LIN {X 0,Y 251.006,Z 606.536,A -85,B 0,C 180,E1 -21636.76,E2 -21636.76} C_VEL
LIN {X 0,Y 251.097,Z 608.017,A -85,B 0,C 180,E1 -21638.716,E2 -21638.716} C_VEL
LIN {X 0,Y 252.117,Z 613.04,A -85,B 0,C 180,E1 -21642.131,E2 -21642.131} C_VEL
LIN {X 0,Y 253.267,Z 618.473,A -85,B 0,C 180,E1 -21644.407,E2 -21644.407} C_VEL
LIN {X 0,Y 253.959,Z 622.03,A -85,B 0,C 180,E1 -21645.519,E2 -21645.519} C_VEL
LIN {X 0,Y 253.455,Z 627.065,A -85,B 0,C 180,E1 -21645.978,E2 -21645.978} C_VEL
LIN {X 0,Y 248.316,Z 655.922,A -85,B 0,C 180,E1 -21647.215,E2 -21647.215} C_VEL
LIN {X 0,Y 244.438,Z 670.422,A -85,B 0,C 180,E1 -21648.052,E2 -21648.052} C_VEL
LIN {X 0,Y 239.958,Z 683.391,A -85,B 0,C 180,E1 -21649.057,E2 -21649.057} C_VEL
LIN {X 0,Y 234.475,Z 696.377,A -85,B 0,C 180,E1 -21650.438,E2 -21650.438} C_VEL
LIN {X 0,Y 229.245,Z 707.125,A -85,B 0,C 180,E1 -21651.906,E2 -21651.906} C_VEL
LIN {X 0,Y 224.326,Z 716.094,A -85,B 0,C 180,E1 -21653.47,E2 -21653.47} C_VEL
LIN {X 0,Y 218.242,Z 725.992,A -85,B 0,C 180,E1 -21655.699,E2 -21655.699} C_VEL
LIN {X 0,Y 212.71,Z 734.271,A -85,B 0,C 180,E1 -21658.087,E2 -21658.087} C_VEL
LIN {X 0,Y 207.703,Z 741.106,A -85,B 0,C 180,E1 -21660.619,E2 -21660.619} C_VEL
LIN {X 0,Y 203.369,Z 746.721,A -85,B 0,C 180,E1 -21663.305,E2 -21663.305} C_VEL
LIN {X 0,Y 199.028,Z 752.063,A -85,B 0,C 180,E1 -21666.65,E2 -21666.65} C_VEL
LIN {X 0,Y 194.978,Z 756.672,A -85,B 0,C 180,E1 -21670.798,E2 -21670.798} C_VEL
LIN {X 0,Y 193.548,Z 761.471,A -85,B 0,C 180,E1 -21673.113,E2 -21673.113} C_VEL
LIN {X 0,Y 191.946,Z 766.73,A -85,B 0,C 180,E1 -21676.232,E2 -21676.232} C_VEL
LIN {X 0,Y 190.963,Z 770.807,A -85,B 0,C 180,E1 -21679.397,E2 -21679.397} C_VEL
LIN {X 0,Y 190.551,Z 772.919,A -85,B 0,C 180,E1 -21681.516,E2 -21681.516} C_VEL
LIN {X 0,Y 190.296,Z 774.58,A -85,B 0,C 180,E1 -21683.639,E2 -21683.639} C_VEL
LIN {X 0,Y 190.173,Z 776.055,A -85,B 0,C 180,E1 -21686.202,E2 -21686.202} C_VEL
LIN {X 0,Y 190.278,Z 777.079,A -85,B 0,C 180,E1 -21690,E2 -21690} C_VEL
LIN {X 0,Y 190.186,Z 776.786,A -85,B 0,C 180,E1 -21693.856,E2 -21693.856} C_VEL
LIN {X 0,Y 190.295,Z 775.895,A -85,B 0,C 180,E1 -21696.361,E2 -21696.361} C_VEL
LIN {X 0,Y 191.029,Z 773.025,A -85,B 0,C 180,E1 -21700.6,E2 -21700.6} C_VEL
LIN {X 0,Y 192.051,Z 769.734,A -85,B 0,C 180,E1 -21703.76,E2 -21703.76} C_VEL
LIN {X 0,Y 193.68,Z 765.366,A -85,B 0,C 180,E1 -21706.875,E2 -21706.875} C_VEL
LIN {X 0,Y 195.856,Z 759.795,A -85,B 0,C 180,E1 -21709.931,E2 -21709.931} C_VEL
LIN {X 0,Y 198.526,Z 752.813,A -85,B 0,C 180,E1 -21712.917,E2 -21712.917} C_VEL
LIN {X 0,Y 201.626,Z 744.079,A -85,B 0,C 180,E1 -21715.83,E2 -21715.83} C_VEL
LIN {X 0,Y 204.75,Z 735.123,A -85,B 0,C 180,E1 -21718.161,E2 -21718.161} C_VEL
LIN {X 0,Y 207.877,Z 725.227,A -85,B 0,C 180,E1 -21720.191,E2 -21720.191} C_VEL
LIN {X 0,Y 210.84,Z 714.228,A -85,B 0,C 180,E1 -21721.948,E2 -21721.948} C_VEL
LIN {X 0,Y 213.609,Z 701.918,A -85,B 0,C 180,E1 -21723.441,E2 -21723.441} C_VEL
LIN {X 0,Y 215.784,Z 689.342,A -85,B 0,C 180,E1 -21724.534,E2 -21724.534} C_VEL
LIN {X 0,Y 217.443,Z 676.109,A -85,B 0,C 180,E1 -21725.291,E2 -21725.291} C_VEL
LIN {X 0,Y 218.773,Z 651.985,A -85,B 0,C 180,E1 -21726.098,E2 -21726.098} C_VEL
LIN {X 0,Y 220.357,Z 618.663,A -85,B 0,C 180,E1 -21727.123,E2 -21727.123} C_VEL
LIN {X 0,Y 218.124,Z 593.995,A -85,B 0,C 180,E1 -21728.604,E2 -21728.604} C_VEL
LIN {X 0,Y 217.001,Z 585.988,A -85,B 0,C 180,E1 -21729.186,E2 -21729.186} C_VEL
LIN {X 0,Y 210.259,Z 568.029,A -85,B 0,C 180,E1 -21731.555,E2 -21731.555} C_VEL
LIN {X 0,Y 203.577,Z 557.24,A -85,B 0,C 180,E1 -21733.891,E2 -21733.891} C_VEL
LIN {X 0,Y 198.403,Z 546.983,A -85,B 0,C 180,E1 -21737.699,E2 -21737.699} C_VEL
LIN {X 0,Y 194.86,Z 539.815,A -85,B 0,C 180,E1 -21740.727,E2 -21740.727} C_VEL
LIN {X 0,Y 193.325,Z 537.896,A -85,B 0,C 180,E1 -21741.83,E2 -21741.83} C_VEL
LIN {X 0,Y 192.59,Z 535.475,A -85,B 0,C 180,E1 -21742.857,E2 -21742.857} C_VEL
LIN {X 0,Y 192.605,Z 535.485,A -85,B 0,C 180,E1 -21747.059,E2 -21747.059} C_VEL
LIN {X 0,Y 192.661,Z 535.48,A -85,B 0,C 180,E1 -21751.692,E2 -21751.692} C_VEL
LIN {X 0,Y 192.681,Z 535.45,A -85,B 0,C 180,E1 -21756.346,E2 -21756.346} C_VEL
LIN {X 0,Y 192.727,Z 535.456,A -85,B 0,C 180,E1 -21761.458,E2 -21761.458} C_VEL
LIN {X 0,Y 192.847,Z 535.464,A -85,B 0,C 180,E1 -21767.37,E2 -21767.37} C_VEL
LIN {X 0,Y 193.057,Z 535.397,A -85,B 0,C 180,E1 -21771.628,E2 -21771.628} C_VEL
LIN {X 0,Y 193.26,Z 535.387,A -85,B 0,C 180,E1 -21777.916,E2 -21777.916} C_VEL
LIN {X 0,Y 193.439,Z 535.348,A -85,B 0,C 180,E1 -21780,E2 -21780} C_VEL
LIN {X 0,Y 192.973,Z 535.448,A -85,B 0,C 180,E1 -21784.178,E2 -21784.178} C_VEL
LIN {X 0,Y 193.033,Z 535.401,A -85,B 0,C 180,E1 -21788.374,E2 -21788.374} C_VEL
LIN {X 0,Y 192.797,Z 535.471,A -85,B 0,C 180,E1 -21792.634,E2 -21792.634} C_VEL
LIN {X 0,Y 192.766,Z 535.44,A -85,B 0,C 180,E1 -21796.959,E2 -21796.959} C_VEL
LIN {X 0,Y 192.638,Z 535.474,A -85,B 0,C 180,E1 -21801.398,E2 -21801.398} C_VEL
LIN {X 0,Y 192.662,Z 535.461,A -85,B 0,C 180,E1 -21804.225,E2 -21804.225} C_VEL
LIN {X 0,Y 192.648,Z 535.466,A -85,B 0,C 180,E1 -21808.893,E2 -21808.893} C_VEL
LIN {X 0,Y 192.575,Z 535.587,A -85,B 0,C 180,E1 -21813.976,E2 -21813.976} C_VEL
LIN {X 0,Y 195.327,Z 542.149,A -85,B 0,C 180,E1 -21817.711,E2 -21817.711} C_VEL
LIN {X 0,Y 198.136,Z 549.33,A -85,B 0,C 180,E1 -21821.37,E2 -21821.37} C_VEL
LIN {X 0,Y 199.487,Z 552.841,A -85,B 0,C 180,E1 -21822.961,E2 -21822.961} C_VEL
LIN {X 0,Y 206.186,Z 563.78,A -85,B 0,C 180,E1 -21825.381,E2 -21825.381} C_VEL
LIN {X 0,Y 213.008,Z 576.443,A -85,B 0,C 180,E1 -21827.668,E2 -21827.668} C_VEL
LIN {X 0,Y 218.113,Z 587.579,A -85,B 0,C 180,E1 -21829.308,E2 -21829.308} C_VEL
LIN {X 0,Y 221.247,Z 595.251,A -85,B 0,C 180,E1 -21830.294,E2 -21830.294} C_VEL
LIN {X 0,Y 221.814,Z 599.859,A -85,B 0,C 180,E1 -21830.598,E2 -21830.598} C_VEL
LIN {X 0,Y 218.375,Z 664.631,A -85,B 0,C 180,E1 -21832.595,E2 -21832.595} C_VEL
LIN {X 0,Y 216.972,Z 677.691,A -85,B 0,C 180,E1 -21833.33,E2 -21833.33} C_VEL
LIN {X 0,Y 214.979,Z 690.5,A -85,B 0,C 180,E1 -21834.43,E2 -21834.43} C_VEL
LIN {X 0,Y 212.604,Z 702.221,A -85,B 0,C 180,E1 -21835.809,E2 -21835.809} C_VEL
LIN {X 0,Y 209.799,Z 713.578,A -85,B 0,C 180,E1 -21837.591,E2 -21837.591} C_VEL
LIN {X 0,Y 206.655,Z 723.812,A -85,B 0,C 180,E1 -21839.611,E2 -21839.611} C_VEL
LIN {X 0,Y 203.821,Z 732.188,A -85,B 0,C 180,E1 -21841.699,E2 -21841.699} C_VEL
LIN {X 0,Y 200.994,Z 739.9,A -85,B 0,C 180,E1 -21844.083,E2 -21844.083} C_VEL
LIN {X 0,Y 198.07,Z 747.411,A -85,B 0,C 180,E1 -21847.027,E2 -21847.027} C_VEL
LIN {X 0,Y 195.739,Z 753.428,A -85,B 0,C 180,E1 -21850.057,E2 -21850.057} C_VEL
LIN {X 0,Y 193.716,Z 758.18,A -85,B 0,C 180,E1 -21853.128,E2 -21853.128} C_VEL
LIN {X 0,Y 192.194,Z 761.808,A -85,B 0,C 180,E1 -21856.25,E2 -21856.25} C_VEL
LIN {X 0,Y 191.192,Z 764.418,A -85,B 0,C 180,E1 -21859.409,E2 -21859.409} C_VEL
LIN {X 0,Y 190.711,Z 765.641,A -85,B 0,C 180,E1 -21861.524,E2 -21861.524} C_VEL
LIN {X 0,Y 190.381,Z 766.46,A -85,B 0,C 180,E1 -21863.642,E2 -21863.642} C_VEL
LIN {X 0,Y 190.235,Z 766.859,A -85,B 0,C 180,E1 -21865.946,E2 -21865.946} C_VEL
LIN {X 0,Y 190.278,Z 766.481,A -85,B 0,C 180,E1 -21870,E2 -21870} C_VEL
LIN {X 0,Y 190.404,Z 765.703,A -85,B 0,C 180,E1 -21872.115,E2 -21872.115} C_VEL
LIN {X 0,Y 190.718,Z 764.501,A -85,B 0,C 180,E1 -21874.226,E2 -21874.226} C_VEL
LIN {X 0,Y 191.346,Z 761.945,A -85,B 0,C 180,E1 -21877.385,E2 -21877.385} C_VEL
LIN {X 0,Y 192.355,Z 758.383,A -85,B 0,C 180,E1 -21880.526,E2 -21880.526} C_VEL
LIN {X 0,Y 193.849,Z 753.714,A -85,B 0,C 180,E1 -21883.63,E2 -21883.63} C_VEL
LIN {X 0,Y 196.246,Z 746.703,A -85,B 0,C 180,E1 -21887.184,E2 -21887.184} C_VEL
LIN {X 0,Y 198.735,Z 739.013,A -85,B 0,C 180,E1 -21890.169,E2 -21890.169} C_VEL
LIN {X 0,Y 201.736,Z 729.422,A -85,B 0,C 180,E1 -21893.074,E2 -21893.074} C_VEL
LIN {X 0,Y 204.231,Z 720.549,A -85,B 0,C 180,E1 -21895.204,E2 -21895.204} C_VEL
LIN {X 0,Y 207.06,Z 709.544,A -85,B 0,C 180,E1 -21897.271,E2 -21897.271} C_VEL
LIN {X 0,Y 209.433,Z 698.253,A -85,B 0,C 180,E1 -21898.931,E2 -21898.931} C_VEL
LIN {X 0,Y 211.508,Z 686.162,A -85,B 0,C 180,E1 -21900.266,E2 -21900.266} C_VEL
LIN {X 0,Y 213.1,Z 672.833,A -85,B 0,C 180,E1 -21901.314,E2 -21901.314} C_VEL
LIN {X 0,Y 214.137,Z 659.825,A -85,B 0,C 180,E1 -21901.951,E2 -21901.951} C_VEL
LIN {X 0,Y 217.094,Z 596.079,A -85,B 0,C 180,E1 -21903.944,E2 -21903.944} C_VEL
LIN {X 0,Y 215.869,Z 587.883,A -85,B 0,C 180,E1 -21904.501,E2 -21904.501} C_VEL
LIN {X 0,Y 210.833,Z 575.542,A -85,B 0,C 180,E1 -21906.003,E2 -21906.003} C_VEL
LIN {X 0,Y 204.574,Z 562.896,A -85,B 0,C 180,E1 -21907.9,E2 -21907.9} C_VEL
LIN {X 0,Y 198.85,Z 552.42,A -85,B 0,C 180,E1 -21909.753,E2 -21909.753} C_VEL
LIN {X 0,Y 196.161,Z 544.735,A -85,B 0,C 180,E1 -21913.074,E2 -21913.074} C_VEL
LIN {X 0,Y 195.594,Z 544.317,A -85,B 0,C 180,E1 -21913.407,E2 -21913.407} C_VEL
LIN {X 0,Y 203.792,Z 567.858,A -85,B 0,C 180,E1 -21915.364,E2 -21915.364} C_VEL
LIN {X 0,Y 200.422,Z 631.067,A -85,B 0,C 180,E1 -21918.682,E2 -21918.682} C_VEL
LIN {X 0,Y 199.667,Z 643.626,A -85,B 0,C 180,E1 -21919.7,E2 -21919.7} C_VEL
LIN {X 0,Y 198.409,Z 656.384,A -85,B 0,C 180,E1 -21921.095,E2 -21921.095} C_VEL
LIN {X 0,Y 196.986,Z 669.363,A -85,B 0,C 180,E1 -21922.982,E2 -21922.982} C_VEL
LIN {X 0,Y 195.719,Z 680.038,A -85,B 0,C 180,E1 -21924.932,E2 -21924.932} C_VEL
LIN {X 0,Y 194.244,Z 691.062,A -85,B 0,C 180,E1 -21927.438,E2 -21927.438} C_VEL
LIN {X 0,Y 192.906,Z 701.42,A -85,B 0,C 180,E1 -21930.361,E2 -21930.361} C_VEL
LIN {X 0,Y 191.938,Z 709.902,A -85,B 0,C 180,E1 -21933.349,E2 -21933.349} C_VEL
LIN {X 0,Y 191.252,Z 716.415,A -85,B 0,C 180,E1 -21936.157,E2 -21936.157} C_VEL
LIN {X 0,Y 190.736,Z 722.668,A -85,B 0,C 180,E1 -21939.509,E2 -21939.509} C_VEL
LIN {X 0,Y 190.549,Z 727.537,A -85,B 0,C 180,E1 -21942.838,E2 -21942.838} C_VEL
LIN {X 0,Y 190.823,Z 731.207,A -85,B 0,C 180,E1 -21946.149,E2 -21946.149} C_VEL
LIN {X 0,Y 191.538,Z 733.793,A -85,B 0,C 180,E1 -21949.428,E2 -21949.428} C_VEL
LIN {X 0,Y 192.288,Z 734.962,A -85,B 0,C 180,E1 -21951.593,E2 -21951.593} C_VEL
LIN {X 0,Y 193.219,Z 735.671,A -85,B 0,C 180,E1 -21953.735,E2 -21953.735} C_VEL
LIN {X 0,Y 194.384,Z 735.979,A -85,B 0,C 180,E1 -21955.853,E2 -21955.853} C_VEL
LIN {X 0,Y 196.797,Z 735.588,A -85,B 0,C 180,E1 -21959.229,E2 -21959.229} C_VEL
LIN {X 0,Y 199.268,Z 734.41,A -85,B 0,C 180,E1 -21962.021,E2 -21962.021} C_VEL
LIN {X 0,Y 201.385,Z 733.053,A -85,B 0,C 180,E1 -21964.002,E2 -21964.002} C_VEL
LIN {X 0,Y 205.459,Z 729.745,A -85,B 0,C 180,E1 -21967.27,E2 -21967.27} C_VEL
LIN {X 0,Y 210.465,Z 724.746,A -85,B 0,C 180,E1 -21970.583,E2 -21970.583} C_VEL
LIN {X 0,Y 216.064,Z 718.252,A -85,B 0,C 180,E1 -21973.64,E2 -21973.64} C_VEL
LIN {X 0,Y 221.287,Z 711.186,A -85,B 0,C 180,E1 -21976.134,E2 -21976.134} C_VEL
LIN {X 0,Y 226.988,Z 702.456,A -85,B 0,C 180,E1 -21978.503,E2 -21978.503} C_VEL
LIN {X 0,Y 232.218,Z 693.181,A -85,B 0,C 180,E1 -21980.46,E2 -21980.46} C_VEL
LIN {X 0,Y 234.395,Z 688.815,A -85,B 0,C 180,E1 -21981.23,E2 -21981.23} C_VEL
LIN {X 0,Y 236.313,Z 684.404,A -85,B 0,C 180,E1 -21982.07,E2 -21982.07} C_VEL
LIN {X 0,Y 238.302,Z 677.52,A -85,B 0,C 180,E1 -21983.734,E2 -21983.734} C_VEL
LIN {X 0,Y 240.139,Z 670.289,A -85,B 0,C 180,E1 -21985.28,E2 -21985.28} C_VEL
LIN {X 0,Y 241.666,Z 665.344,A -85,B 0,C 180,E1 -21985.936,E2 -21985.936} C_VEL
LIN {X 0,Y 245.716,Z 652.137,A -85,B 0,C 180,E1 -21987.063,E2 -21987.063} C_VEL
LIN {X 0,Y 248.489,Z 640.109,A -85,B 0,C 180,E1 -21987.813,E2 -21987.813} C_VEL
LIN {X 0,Y 252.626,Z 616.909,A -85,B 0,C 180,E1 -21988.85,E2 -21988.85} C_VEL
LIN {X 0,Y 251.193,Z 614.269,A -85,B 0,C 180,E1 -21991.022,E2 -21991.022} C_VEL
LIN {X 0,Y 250.108,Z 613.02,A -85,B 0,C 180,E1 -21993.377,E2 -21993.377} C_VEL
LIN {X 0,Y 249.533,Z 613.107,A -85,B 0,C 180,E1 -21995.798,E2 -21995.798} C_VEL
LIN {X 0,Y 249.495,Z 614.676,A -85,B 0,C 180,E1 -21998.295,E2 -21998.295} C_VEL
LIN {X 0,Y 250.173,Z 619.582,A -85,B 0,C 180,E1 -22001.613,E2 -22001.613} C_VEL
LIN {X 0,Y 251.095,Z 624.646,A -85,B 0,C 180,E1 -22003.755,E2 -22003.755} C_VEL
LIN {X 0,Y 251.331,Z 626.487,A -85,B 0,C 180,E1 -22004.326,E2 -22004.326} C_VEL
LIN {X 0,Y 250.759,Z 630.367,A -85,B 0,C 180,E1 -22004.567,E2 -22004.567} C_VEL
LIN {X 0,Y 246.269,Z 654.434,A -85,B 0,C 180,E1 -22005.588,E2 -22005.588} C_VEL
LIN {X 0,Y 242.488,Z 668.206,A -85,B 0,C 180,E1 -22006.359,E2 -22006.359} C_VEL
LIN {X 0,Y 238.113,Z 680.483,A -85,B 0,C 180,E1 -22007.247,E2 -22007.247} C_VEL
LIN {X 0,Y 232.965,Z 692.693,A -85,B 0,C 180,E1 -22008.42,E2 -22008.42} C_VEL
LIN {X 0,Y 226.813,Z 704.914,A -85,B 0,C 180,E1 -22009.989,E2 -22009.989} C_VEL
LIN {X 0,Y 221.005,Z 714.949,A -85,B 0,C 180,E1 -22011.677,E2 -22011.677} C_VEL
LIN {X 0,Y 214.571,Z 724.937,A -85,B 0,C 180,E1 -22013.875,E2 -22013.875} C_VEL
LIN {X 0,Y 208.674,Z 733.174,A -85,B 0,C 180,E1 -22016.241,E2 -22016.241} C_VEL
LIN {X 0,Y 202.458,Z 741.076,A -85,B 0,C 180,E1 -22019.202,E2 -22019.202} C_VEL
LIN {X 0,Y 197.082,Z 747.344,A -85,B 0,C 180,E1 -22022.382,E2 -22022.382} C_VEL
LIN {X 0,Y 192.036,Z 752.839,A -85,B 0,C 180,E1 -22026.262,E2 -22026.262} C_VEL
LIN {X 0,Y 188.05,Z 756.968,A -85,B 0,C 180,E1 -22030.345,E2 -22030.345} C_VEL
LIN {X 0,Y 186.738,Z 761.216,A -85,B 0,C 180,E1 -22032.478,E2 -22032.478} C_VEL
LIN {X 0,Y 185.003,Z 766.487,A -85,B 0,C 180,E1 -22035.705,E2 -22035.705} C_VEL
LIN {X 0,Y 183.945,Z 770.576,A -85,B 0,C 180,E1 -22038.987,E2 -22038.987} C_VEL
LIN {X 0,Y 183.515,Z 772.699,A -85,B 0,C 180,E1 -22041.189,E2 -22041.189} C_VEL
LIN {X 0,Y 183.224,Z 774.366,A -85,B 0,C 180,E1 -22043.392,E2 -22043.392} C_VEL
LIN {X 0,Y 183.083,Z 775.99,A -85,B 0,C 180,E1 -22046.43,E2 -22046.43} C_VEL
LIN {X 0,Y 183.184,Z 776.885,A -85,B 0,C 180,E1 -22050,E2 -22050} C_VEL
LIN {X 0,Y 183.099,Z 776.682,A -85,B 0,C 180,E1 -22053.65,E2 -22053.65} C_VEL
LIN {X 0,Y 183.224,Z 775.722,A -85,B 0,C 180,E1 -22056.608,E2 -22056.608} C_VEL
LIN {X 0,Y 184.036,Z 772.863,A -85,B 0,C 180,E1 -22061.007,E2 -22061.007} C_VEL
LIN {X 0,Y 185.124,Z 769.582,A -85,B 0,C 180,E1 -22064.286,E2 -22064.286} C_VEL
LIN {X 0,Y 186.87,Z 765.228,A -85,B 0,C 180,E1 -22067.51,E2 -22067.51} C_VEL
LIN {X 0,Y 189.164,Z 759.67,A -85,B 0,C 180,E1 -22070.668,E2 -22070.668} C_VEL
LIN {X 0,Y 191.536,Z 753.891,A -85,B 0,C 180,E1 -22073.265,E2 -22073.265} C_VEL
LIN {X 0,Y 194.65,Z 745.609,A -85,B 0,C 180,E1 -22076.25,E2 -22076.25} C_VEL
LIN {X 0,Y 197.828,Z 736.995,A -85,B 0,C 180,E1 -22078.658,E2 -22078.658} C_VEL
LIN {X 0,Y 201.385,Z 726.391,A -85,B 0,C 180,E1 -22080.98,E2 -22080.98} C_VEL
LIN {X 0,Y 204.454,Z 715.807,A -85,B 0,C 180,E1 -22082.778,E2 -22082.778} C_VEL
LIN {X 0,Y 207.325,Z 703.947,A -85,B 0,C 180,E1 -22084.301,E2 -22084.301} C_VEL
LIN {X 0,Y 209.664,Z 691.635,A -85,B 0,C 180,E1 -22085.472,E2 -22085.472} C_VEL
LIN {X 0,Y 211.484,Z 678.711,A -85,B 0,C 180,E1 -22086.294,E2 -22086.294} C_VEL
LIN {X 0,Y 212.586,Z 663.23,A -85,B 0,C 180,E1 -22086.891,E2 -22086.891} C_VEL
LIN {X 0,Y 214.742,Z 619.115,A -85,B 0,C 180,E1 -22088.283,E2 -22088.283} C_VEL
LIN {X 0,Y 212.663,Z 595.341,A -85,B 0,C 180,E1 -22089.767,E2 -22089.767} C_VEL
LIN {X 0,Y 211.799,Z 588.832,A -85,B 0,C 180,E1 -22090.254,E2 -22090.254} C_VEL
LIN {X 0,Y 205.673,Z 572.134,A -85,B 0,C 180,E1 -22092.54,E2 -22092.54} C_VEL
LIN {X 0,Y 198.272,Z 560.516,A -85,B 0,C 180,E1 -22095.189,E2 -22095.189} C_VEL
LIN {X 0,Y 196.082,Z 557.012,A -85,B 0,C 180,E1 -22096.119,E2 -22096.119} C_VEL
LIN {X 0,Y 191.992,Z 548.836,A -85,B 0,C 180,E1 -22099.478,E2 -22099.478} C_VEL
LIN {X 0,Y 190.214,Z 545.178,A -85,B 0,C 180,E1 -22101.089,E2 -22101.089} C_VEL
LIN {X 0,Y 188.506,Z 542.674,A -85,B 0,C 180,E1 -22102.455,E2 -22102.455} C_VEL
LIN {X 0,Y 187.902,Z 540.804,A -85,B 0,C 180,E1 -22103.242,E2 -22103.242} C_VEL
LIN {X 0,Y 186.047,Z 538.224,A -85,B 0,C 180,E1 -22104.825,E2 -22104.825} C_VEL
LIN {X 0,Y 185.534,Z 536.37,A -85,B 0,C 180,E1 -22105.691,E2 -22105.691} C_VEL
LIN {X 0,Y 185.579,Z 536.346,A -85,B 0,C 180,E1 -22110.576,E2 -22110.576} C_VEL
LIN {X 0,Y 185.576,Z 536.336,A -85,B 0,C 180,E1 -22115.381,E2 -22115.381} C_VEL
LIN {X 0,Y 185.67,Z 536.339,A -85,B 0,C 180,E1 -22121.134,E2 -22121.134} C_VEL
LIN {X 0,Y 185.759,Z 536.344,A -85,B 0,C 180,E1 -22126.88,E2 -22126.88} C_VEL
LIN {X 0,Y 186.004,Z 536.275,A -85,B 0,C 180,E1 -22131.308,E2 -22131.308} C_VEL
LIN {X 0,Y 186.204,Z 536.266,A -85,B 0,C 180,E1 -22137.837,E2 -22137.837} C_VEL
LIN {X 0,Y 186.403,Z 536.224,A -85,B 0,C 180,E1 -22140,E2 -22140} C_VEL
LIN {X 0,Y 185.92,Z 536.327,A -85,B 0,C 180,E1 -22144.336,E2 -22144.336} C_VEL
LIN {X 0,Y 185.979,Z 536.28,A -85,B 0,C 180,E1 -22148.695,E2 -22148.695} C_VEL
LIN {X 0,Y 185.724,Z 536.347,A -85,B 0,C 180,E1 -22153.124,E2 -22153.124} C_VEL
LIN {X 0,Y 185.713,Z 536.323,A -85,B 0,C 180,E1 -22157.623,E2 -22157.623} C_VEL
LIN {X 0,Y 185.597,Z 536.341,A -85,B 0,C 180,E1 -22162.252,E2 -22162.252} C_VEL
LIN {X 0,Y 185.561,Z 536.369,A -85,B 0,C 180,E1 -22167.033,E2 -22167.033} C_VEL
LIN {X 0,Y 185.567,Z 536.472,A -85,B 0,C 180,E1 -22171.225,E2 -22171.225} C_VEL
LIN {X 0,Y 185.855,Z 537.779,A -85,B 0,C 180,E1 -22171.966,E2 -22171.966} C_VEL
LIN {X 0,Y 188.314,Z 543.037,A -85,B 0,C 180,E1 -22175.343,E2 -22175.343} C_VEL
LIN {X 0,Y 190.843,Z 549.044,A -85,B 0,C 180,E1 -22178.76,E2 -22178.76} C_VEL
LIN {X 0,Y 192.446,Z 553.126,A -85,B 0,C 180,E1 -22180.754,E2 -22180.754} C_VEL
LIN {X 0,Y 199.267,Z 563.834,A -85,B 0,C 180,E1 -22183.453,E2 -22183.453} C_VEL
LIN {X 0,Y 205.495,Z 574.879,A -85,B 0,C 180,E1 -22185.722,E2 -22185.722} C_VEL
LIN {X 0,Y 210.934,Z 585.987,A -85,B 0,C 180,E1 -22187.597,E2 -22187.597} C_VEL
LIN {X 0,Y 215.927,Z 597.982,A -85,B 0,C 180,E1 -22189.268,E2 -22189.268} C_VEL
LIN {X 0,Y 216.242,Z 600.852,A -85,B 0,C 180,E1 -22189.459,E2 -22189.459} C_VEL
LIN {X 0,Y 212.669,Z 665.3,A -85,B 0,C 180,E1 -22191.486,E2 -22191.486} C_VEL
LIN {X 0,Y 211.198,Z 678.141,A -85,B 0,C 180,E1 -22192.231,E2 -22192.231} C_VEL
LIN {X 0,Y 209.216,Z 690.349,A -85,B 0,C 180,E1 -22193.294,E2 -22193.294} C_VEL
LIN {X 0,Y 206.733,Z 702.157,A -85,B 0,C 180,E1 -22194.696,E2 -22194.696} C_VEL
LIN {X 0,Y 203.839,Z 713.573,A -85,B 0,C 180,E1 -22196.521,E2 -22196.521} C_VEL
LIN {X 0,Y 200.562,Z 723.842,A -85,B 0,C 180,E1 -22198.585,E2 -22198.585} C_VEL
LIN {X 0,Y 197.591,Z 732.246,A -85,B 0,C 180,E1 -22200.722,E2 -22200.722} C_VEL
LIN {X 0,Y 194.626,Z 739.981,A -85,B 0,C 180,E1 -22203.169,E2 -22203.169} C_VEL
LIN {X 0,Y 191.525,Z 747.52,A -85,B 0,C 180,E1 -22206.194,E2 -22206.194} C_VEL
LIN {X 0,Y 189.024,Z 753.553,A -85,B 0,C 180,E1 -22209.316,E2 -22209.316} C_VEL
LIN {X 0,Y 186.926,Z 758.319,A -85,B 0,C 180,E1 -22212.496,E2 -22212.496} C_VEL
LIN {X 0,Y 185.277,Z 761.96,A -85,B 0,C 180,E1 -22215.726,E2 -22215.726} C_VEL
LIN {X 0,Y 184.181,Z 764.583,A -85,B 0,C 180,E1 -22219.001,E2 -22219.001} C_VEL
LIN {X 0,Y 183.673,Z 765.812,A -85,B 0,C 180,E1 -22221.196,E2 -22221.196} C_VEL
LIN {X 0,Y 183.319,Z 766.641,A -85,B 0,C 180,E1 -22223.396,E2 -22223.396} C_VEL
LIN {X 0,Y 183.138,Z 767.075,A -85,B 0,C 180,E1 -22226.18,E2 -22226.18} C_VEL
LIN {X 0,Y 183.184,Z 766.681,A -85,B 0,C 180,E1 -22230,E2 -22230} C_VEL
LIN {X 0,Y 183.318,Z 765.914,A -85,B 0,C 180,E1 -22232.197,E2 -22232.197} C_VEL
LIN {X 0,Y 183.644,Z 764.717,A -85,B 0,C 180,E1 -22234.39,E2 -22234.39} C_VEL
LIN {X 0,Y 184.22,Z 762.534,A -85,B 0,C 180,E1 -22237.29,E2 -22237.29} C_VEL
LIN {X 0,Y 185.376,Z 758.624,A -85,B 0,C 180,E1 -22240.927,E2 -22240.927} C_VEL
LIN {X 0,Y 186.97,Z 753.968,A -85,B 0,C 180,E1 -22244.142,E2 -22244.142} C_VEL
LIN {X 0,Y 189.471,Z 746.974,A -85,B 0,C 180,E1 -22247.819,E2 -22247.819} C_VEL
LIN {X 0,Y 192.102,Z 739.305,A -85,B 0,C 180,E1 -22250.897,E2 -22250.897} C_VEL
LIN {X 0,Y 195.22,Z 729.734,A -85,B 0,C 180,E1 -22253.891,E2 -22253.891} C_VEL
LIN {X 0,Y 198.199,Z 719.766,A -85,B 0,C 180,E1 -22256.31,E2 -22256.31} C_VEL
LIN {X 0,Y 201.211,Z 708.54,A -85,B 0,C 180,E1 -22258.417,E2 -22258.417} C_VEL
LIN {X 0,Y 203.523,Z 697.55,A -85,B 0,C 180,E1 -22260.042,E2 -22260.042} C_VEL
LIN {X 0,Y 205.665,Z 685.088,A -85,B 0,C 180,E1 -22261.406,E2 -22261.406} C_VEL
LIN {X 0,Y 207.242,Z 672.034,A -85,B 0,C 180,E1 -22262.426,E2 -22262.426} C_VEL
LIN {X 0,Y 208.285,Z 658.961,A -85,B 0,C 180,E1 -22263.045,E2 -22263.045} C_VEL
LIN {X 0,Y 211.335,Z 597.63,A -85,B 0,C 180,E1 -22264.983,E2 -22264.983} C_VEL
LIN {X 0,Y 210.213,Z 590.16,A -85,B 0,C 180,E1 -22265.518,E2 -22265.518} C_VEL
LIN {X 0,Y 205.221,Z 578.164,A -85,B 0,C 180,E1 -22267.083,E2 -22267.083} C_VEL
LIN {X 0,Y 198.598,Z 564.635,A -85,B 0,C 180,E1 -22269.229,E2 -22269.229} C_VEL
LIN {X 0,Y 193.412,Z 555.568,A -85,B 0,C 180,E1 -22270.989,E2 -22270.989} C_VEL
LIN {X 0,Y 191.659,Z 552.418,A -85,B 0,C 180,E1 -22271.701,E2 -22271.701} C_VEL
LIN {X 0,Y 190.947,Z 550.361,A -85,B 0,C 180,E1 -22272.597,E2 -22272.597} C_VEL
LIN {X 0,Y 190.039,Z 549.424,A -85,B 0,C 180,E1 -22273.185,E2 -22273.185} C_VEL
LIN {X 0,Y 196.819,Z 569.167,A -85,B 0,C 180,E1 -22274.937,E2 -22274.937} C_VEL
LIN {X 0,Y 193.425,Z 631.842,A -85,B 0,C 180,E1 -22278.375,E2 -22278.375} C_VEL
LIN {X 0,Y 192.447,Z 645.892,A -85,B 0,C 180,E1 -22279.578,E2 -22279.578} C_VEL
LIN {X 0,Y 191.027,Z 660.034,A -85,B 0,C 180,E1 -22281.285,E2 -22281.285} C_VEL
LIN {X 0,Y 189.53,Z 672.586,A -85,B 0,C 180,E1 -22283.277,E2 -22283.277} C_VEL
LIN {X 0,Y 188.134,Z 684.169,A -85,B 0,C 180,E1 -22285.618,E2 -22285.618} C_VEL
LIN {X 0,Y 186.725,Z 694.474,A -85,B 0,C 180,E1 -22288.201,E2 -22288.201} C_VEL
LIN {X 0,Y 185.502,Z 703.812,A -85,B 0,C 180,E1 -22291.114,E2 -22291.114} C_VEL
LIN {X 0,Y 184.528,Z 712.914,A -85,B 0,C 180,E1 -22294.629,E2 -22294.629} C_VEL
LIN {X 0,Y 183.803,Z 720.01,A -85,B 0,C 180,E1 -22298.111,E2 -22298.111} C_VEL
LIN {X 0,Y 183.454,Z 726.452,A -85,B 0,C 180,E1 -22302.153,E2 -22302.153} C_VEL
LIN {X 0,Y 183.639,Z 730.563,A -85,B 0,C 180,E1 -22305.595,E2 -22305.595} C_VEL
LIN {X 0,Y 184.302,Z 733.55,A -85,B 0,C 180,E1 -22309.008,E2 -22309.008} C_VEL
LIN {X 0,Y 185.049,Z 734.959,A -85,B 0,C 180,E1 -22311.261,E2 -22311.261} C_VEL
LIN {X 0,Y 187.119,Z 736.54,A -85,B 0,C 180,E1 -22315.691,E2 -22315.691} C_VEL
LIN {X 0,Y 189.76,Z 736.558,A -85,B 0,C 180,E1 -22319.446,E2 -22319.446} C_VEL
LIN {X 0,Y 192.062,Z 735.771,A -85,B 0,C 180,E1 -22322.097,E2 -22322.097} C_VEL
LIN {X 0,Y 194.229,Z 734.7,A -85,B 0,C 180,E1 -22324.15,E2 -22324.15} C_VEL
LIN {X 0,Y 198.53,Z 731.801,A -85,B 0,C 180,E1 -22327.616,E2 -22327.616} C_VEL
LIN {X 0,Y 203.53,Z 727.493,A -85,B 0,C 180,E1 -22330.948,E2 -22330.948} C_VEL
LIN {X 0,Y 208.428,Z 722.549,A -85,B 0,C 180,E1 -22333.652,E2 -22333.652} C_VEL
LIN {X 0,Y 213.817,Z 716.397,A -85,B 0,C 180,E1 -22336.223,E2 -22336.223} C_VEL
LIN {X 0,Y 219.506,Z 708.828,A -85,B 0,C 180,E1 -22338.673,E2 -22338.673} C_VEL
LIN {X 0,Y 225.895,Z 699.043,A -85,B 0,C 180,E1 -22341.04,E2 -22341.04} C_VEL
LIN {X 0,Y 231.457,Z 689.198,A -85,B 0,C 180,E1 -22342.88,E2 -22342.88} C_VEL
LIN {X 0,Y 236.834,Z 677.705,A -85,B 0,C 180,E1 -22344.547,E2 -22344.547} C_VEL
LIN {X 0,Y 241.666,Z 665.344,A -85,B 0,C 180,E1 -22345.936,E2 -22345.936} C_VEL
LIN {X 0,Y 243.187,Z 660.245,A -85,B 0,C 180,E1 -22346.545,E2 -22346.545} C_VEL
LIN {X 0,Y 244.76,Z 652.18,A -85,B 0,C 180,E1 -22347.85,E2 -22347.85} C_VEL
LIN {X 0,Y 246.099,Z 643.883,A -85,B 0,C 180,E1 -22349.043,E2 -22349.043} C_VEL
LIN {X 0,Y 247.077,Z 638.442,A -85,B 0,C 180,E1 -22349.491,E2 -22349.491} C_VEL
LIN {X 0,Y 250.088,Z 622.285,A -85,B 0,C 180,E1 -22350.221,E2 -22350.221} C_VEL
LIN {X 0,Y 249.289,Z 620.914,A -85,B 0,C 180,E1 -22351.623,E2 -22351.623} C_VEL
LIN {X 0,Y 248.454,Z 619.883,A -85,B 0,C 180,E1 -22353.628,E2 -22353.628} C_VEL
LIN {X 0,Y 247.912,Z 620.208,A -85,B 0,C 180,E1 -22356.171,E2 -22356.171} C_VEL
LIN {X 0,Y 247.898,Z 621.634,A -85,B 0,C 180,E1 -22358.125,E2 -22358.125} C_VEL
LIN {X 0,Y 248.339,Z 626.069,A -85,B 0,C 180,E1 -22361.076,E2 -22361.076} C_VEL
LIN {X 0,Y 248.972,Z 630.487,A -85,B 0,C 180,E1 -22362.966,E2 -22362.966} C_VEL
LIN {X 0,Y 244.341,Z 653.847,A -85,B 0,C 180,E1 -22363.978,E2 -22363.978} C_VEL
LIN {X 0,Y 240.611,Z 666.877,A -85,B 0,C 180,E1 -22364.67,E2 -22364.67} C_VEL
LIN {X 0,Y 235.889,Z 679.789,A -85,B 0,C 180,E1 -22365.561,E2 -22365.561} C_VEL
LIN {X 0,Y 230.519,Z 691.858,A -85,B 0,C 180,E1 -22366.689,E2 -22366.689} C_VEL
LIN {X 0,Y 224.087,Z 703.942,A -85,B 0,C 180,E1 -22368.207,E2 -22368.207} C_VEL
LIN {X 0,Y 217.983,Z 714.061,A -85,B 0,C 180,E1 -22369.849,E2 -22369.849} C_VEL
LIN {X 0,Y 211.162,Z 723.981,A -85,B 0,C 180,E1 -22371.996,E2 -22371.996} C_VEL
LIN {X 0,Y 203.893,Z 733.46,A -85,B 0,C 180,E1 -22374.736,E2 -22374.736} C_VEL
LIN {X 0,Y 197.327,Z 741.078,A -85,B 0,C 180,E1 -22377.708,E2 -22377.708} C_VEL
LIN {X 0,Y 190.84,Z 747.931,A -85,B 0,C 180,E1 -22381.397,E2 -22381.397} C_VEL
LIN {X 0,Y 186.747,Z 751.909,A -85,B 0,C 180,E1 -22384.356,E2 -22384.356} C_VEL
LIN {X 0,Y 181.854,Z 756.211,A -85,B 0,C 180,E1 -22389.055,E2 -22389.055} C_VEL
LIN {X 0,Y 181.348,Z 756.707,A -85,B 0,C 180,E1 -22389.587,E2 -22389.587} C_VEL
LIN {X 0,Y 179.277,Z 762.857,A -85,B 0,C 180,E1 -22392.902,E2 -22392.902} C_VEL
LIN {X 0,Y 177.655,Z 767.722,A -85,B 0,C 180,E1 -22396.27,E2 -22396.27} C_VEL
LIN {X 0,Y 176.685,Z 771.454,A -85,B 0,C 180,E1 -22399.689,E2 -22399.689} C_VEL
LIN {X 0,Y 176.148,Z 774.151,A -85,B 0,C 180,E1 -22403.126,E2 -22403.126} C_VEL
LIN {X 0,Y 175.995,Z 775.925,A -85,B 0,C 180,E1 -22406.681,E2 -22406.681} C_VEL
LIN {X 0,Y 176.091,Z 776.692,A -85,B 0,C 180,E1 -22410,E2 -22410} C_VEL
LIN {X 0,Y 175.995,Z 776.6,A -85,B 0,C 180,E1 -22413.32,E2 -22413.32} C_VEL
LIN {X 0,Y 176.149,Z 775.548,A -85,B 0,C 180,E1 -22416.874,E2 -22416.874} C_VEL
LIN {X 0,Y 177.031,Z 772.7,A -85,B 0,C 180,E1 -22421.449,E2 -22421.449} C_VEL
LIN {X 0,Y 178.199,Z 769.431,A -85,B 0,C 180,E1 -22424.853,E2 -22424.853} C_VEL
LIN {X 0,Y 180.091,Z 765.09,A -85,B 0,C 180,E1 -22428.191,E2 -22428.191} C_VEL
LIN {X 0,Y 182.521,Z 759.546,A -85,B 0,C 180,E1 -22431.456,E2 -22431.456} C_VEL
LIN {X 0,Y 185.465,Z 752.61,A -85,B 0,C 180,E1 -22434.634,E2 -22434.634} C_VEL
LIN {X 0,Y 188.908,Z 743.916,A -85,B 0,C 180,E1 -22437.712,E2 -22437.712} C_VEL
LIN {X 0,Y 192.684,Z 734.035,A -85,B 0,C 180,E1 -22440.402,E2 -22440.402} C_VEL
LIN {X 0,Y 196.098,Z 723.926,A -85,B 0,C 180,E1 -22442.519,E2 -22442.519} C_VEL
LIN {X 0,Y 199.297,Z 712.728,A -85,B 0,C 180,E1 -22444.347,E2 -22444.347} C_VEL
LIN {X 0,Y 202.169,Z 701.106,A -85,B 0,C 180,E1 -22445.763,E2 -22445.763} C_VEL
LIN {X 0,Y 204.545,Z 688.329,A -85,B 0,C 180,E1 -22446.884,E2 -22446.884} C_VEL
LIN {X 0,Y 206.284,Z 674.82,A -85,B 0,C 180,E1 -22447.67,E2 -22447.67} C_VEL
LIN {X 0,Y 209.267,Z 619.978,A -85,B 0,C 180,E1 -22449.476,E2 -22449.476} C_VEL
LIN {X 0,Y 207.307,Z 596.672,A -85,B 0,C 180,E1 -22450.989,E2 -22450.989} C_VEL
LIN {X 0,Y 206.504,Z 591.153,A -85,B 0,C 180,E1 -22451.442,E2 -22451.442} C_VEL
LIN {X 0,Y 201.211,Z 576.412,A -85,B 0,C 180,E1 -22453.545,E2 -22453.545} C_VEL
LIN {X 0,Y 194.309,Z 565.414,A -85,B 0,C 180,E1 -22456.155,E2 -22456.155} C_VEL
LIN {X 0,Y 188.646,Z 556.8,A -85,B 0,C 180,E1 -22458.603,E2 -22458.603} C_VEL
LIN {X 0,Y 185.08,Z 549.647,A -85,B 0,C 180,E1 -22461.899,E2 -22461.899} C_VEL
LIN {X 0,Y 183.803,Z 547.681,A -85,B 0,C 180,E1 -22462.998,E2 -22462.998} C_VEL
LIN {X 0,Y 183.349,Z 546.303,A -85,B 0,C 180,E1 -22463.604,E2 -22463.604} C_VEL
LIN {X 0,Y 180.076,Z 540.857,A -85,B 0,C 180,E1 -22466.881,E2 -22466.881} C_VEL
LIN {X 0,Y 178.655,Z 538.068,A -85,B 0,C 180,E1 -22468.585,E2 -22468.585} C_VEL
LIN {X 0,Y 178.491,Z 537.224,A -85,B 0,C 180,E1 -22469.048,E2 -22469.048} C_VEL
LIN {X 0,Y 178.499,Z 537.225,A -85,B 0,C 180,E1 -22474.336,E2 -22474.336} C_VEL
LIN {X 0,Y 178.52,Z 537.245,A -85,B 0,C 180,E1 -22479.249,E2 -22479.249} C_VEL
LIN {X 0,Y 178.645,Z 537.205,A -85,B 0,C 180,E1 -22481.656,E2 -22481.656} C_VEL
LIN {X 0,Y 178.676,Z 537.217,A -85,B 0,C 180,E1 -22486.35,E2 -22486.35} C_VEL
LIN {X 0,Y 178.934,Z 537.157,A -85,B 0,C 180,E1 -22490.961,E2 -22490.961} C_VEL
LIN {X 0,Y 179.15,Z 537.145,A -85,B 0,C 180,E1 -22497.752,E2 -22497.752} C_VEL
LIN {X 0,Y 179.366,Z 537.1,A -85,B 0,C 180,E1 -22500.001,E2 -22500.001} C_VEL
LIN {X 0,Y 178.867,Z 537.206,A -85,B 0,C 180,E1 -22504.508,E2 -22504.508} C_VEL
LIN {X 0,Y 178.908,Z 537.161,A -85,B 0,C 180,E1 -22509.041,E2 -22509.041} C_VEL
LIN {X 0,Y 178.654,Z 537.218,A -85,B 0,C 180,E1 -22513.653,E2 -22513.653} C_VEL
LIN {X 0,Y 178.636,Z 537.228,A -85,B 0,C 180,E1 -22519.231,E2 -22519.231} C_VEL
LIN {X 0,Y 178.533,Z 537.227,A -85,B 0,C 180,E1 -22525.125,E2 -22525.125} C_VEL
LIN {X 0,Y 178.511,Z 537.302,A -85,B 0,C 180,E1 -22527.874,E2 -22527.874} C_VEL
LIN {X 0,Y 180.399,Z 541.471,A -85,B 0,C 180,E1 -22531.012,E2 -22531.012} C_VEL
LIN {X 0,Y 183.93,Z 549.716,A -85,B 0,C 180,E1 -22536.32,E2 -22536.32} C_VEL
LIN {X 0,Y 185.435,Z 553.355,A -85,B 0,C 180,E1 -22538.275,E2 -22538.275} C_VEL
LIN {X 0,Y 192.58,Z 564.308,A -85,B 0,C 180,E1 -22541.41,E2 -22541.41} C_VEL
LIN {X 0,Y 198.217,Z 573.882,A -85,B 0,C 180,E1 -22543.654,E2 -22543.654} C_VEL
LIN {X 0,Y 204.383,Z 585.894,A -85,B 0,C 180,E1 -22545.95,E2 -22545.95} C_VEL
LIN {X 0,Y 210.165,Z 599.33,A -85,B 0,C 180,E1 -22548.008,E2 -22548.008} C_VEL
LIN {X 0,Y 210.772,Z 601.199,A -85,B 0,C 180,E1 -22548.234,E2 -22548.234} C_VEL
LIN {X 0,Y 207.148,Z 664.629,A -85,B 0,C 180,E1 -22550.26,E2 -22550.26} C_VEL
LIN {X 0,Y 205.715,Z 677.151,A -85,B 0,C 180,E1 -22550.959,E2 -22550.959} C_VEL
LIN {X 0,Y 203.608,Z 689.874,A -85,B 0,C 180,E1 -22552.061,E2 -22552.061} C_VEL
LIN {X 0,Y 200.857,Z 702.558,A -85,B 0,C 180,E1 -22553.589,E2 -22553.589} C_VEL
LIN {X 0,Y 197.954,Z 713.569,A -85,B 0,C 180,E1 -22555.387,E2 -22555.387} C_VEL
LIN {X 0,Y 194.526,Z 723.872,A -85,B 0,C 180,E1 -22557.493,E2 -22557.493} C_VEL
LIN {X 0,Y 191.419,Z 732.304,A -85,B 0,C 180,E1 -22559.68,E2 -22559.68} C_VEL
LIN {X 0,Y 188.289,Z 740.062,A -85,B 0,C 180,E1 -22562.189,E2 -22562.189} C_VEL
LIN {X 0,Y 185,Z 747.629,A -85,B 0,C 180,E1 -22565.3,E2 -22565.3} C_VEL
LIN {X 0,Y 182.349,Z 753.678,A -85,B 0,C 180,E1 -22568.523,E2 -22568.523} C_VEL
LIN {X 0,Y 180.158,Z 758.458,A -85,B 0,C 180,E1 -22571.816,E2 -22571.816} C_VEL
LIN {X 0,Y 178.355,Z 762.114,A -85,B 0,C 180,E1 -22575.16,E2 -22575.16} C_VEL
LIN {X 0,Y 177.192,Z 764.748,A -85,B 0,C 180,E1 -22578.562,E2 -22578.562} C_VEL
LIN {X 0,Y 176.636,Z 765.983,A -85,B 0,C 180,E1 -22580.843,E2 -22580.843} C_VEL
LIN {X 0,Y 176.254,Z 766.821,A -85,B 0,C 180,E1 -22583.13,E2 -22583.13} C_VEL
LIN {X 0,Y 176.047,Z 767.288,A -85,B 0,C 180,E1 -22586.415,E2 -22586.415} C_VEL
LIN {X 0,Y 176.092,Z 766.88,A -85,B 0,C 180,E1 -22590,E2 -22590} C_VEL
LIN {X 0,Y 176.234,Z 766.125,A -85,B 0,C 180,E1 -22592.285,E2 -22592.285} C_VEL
LIN {X 0,Y 176.575,Z 764.934,A -85,B 0,C 180,E1 -22594.566,E2 -22594.566} C_VEL
LIN {X 0,Y 177.113,Z 763.046,A -85,B 0,C 180,E1 -22597.236,E2 -22597.236} C_VEL
LIN {X 0,Y 178.427,Z 758.865,A -85,B 0,C 180,E1 -22601.358,E2 -22601.358} C_VEL
LIN {X 0,Y 180.116,Z 754.221,A -85,B 0,C 180,E1 -22604.692,E2 -22604.692} C_VEL
LIN {X 0,Y 182.714,Z 747.243,A -85,B 0,C 180,E1 -22608.501,E2 -22608.501} C_VEL
LIN {X 0,Y 185.503,Z 739.598,A -85,B 0,C 180,E1 -22611.677,E2 -22611.677} C_VEL
LIN {X 0,Y 188.76,Z 730.046,A -85,B 0,C 180,E1 -22614.762,E2 -22614.762} C_VEL
LIN {X 0,Y 191.892,Z 720.112,A -85,B 0,C 180,E1 -22617.245,E2 -22617.245} C_VEL
LIN {X 0,Y 195.012,Z 708.918,A -85,B 0,C 180,E1 -22619.407,E2 -22619.407} C_VEL
LIN {X 0,Y 197.349,Z 698.334,A -85,B 0,C 180,E1 -22621.022,E2 -22621.022} C_VEL
LIN {X 0,Y 199.47,Z 686.835,A -85,B 0,C 180,E1 -22622.349,E2 -22622.349} C_VEL
LIN {X 0,Y 201.216,Z 673.52,A -85,B 0,C 180,E1 -22623.448,E2 -22623.448} C_VEL
LIN {X 0,Y 202.39,Z 660.24,A -85,B 0,C 180,E1 -22624.126,E2 -22624.126} C_VEL
LIN {X 0,Y 205.549,Z 597.938,A -85,B 0,C 180,E1 -22626.154,E2 -22626.154} C_VEL
LIN {X 0,Y 204.743,Z 592.879,A -85,B 0,C 180,E1 -22626.546,E2 -22626.546} C_VEL
LIN {X 0,Y 200.051,Z 581.517,A -85,B 0,C 180,E1 -22628.105,E2 -22628.105} C_VEL
LIN {X 0,Y 193.977,Z 568.941,A -85,B 0,C 180,E1 -22630.189,E2 -22630.189} C_VEL
LIN {X 0,Y 188.533,Z 559.289,A -85,B 0,C 180,E1 -22632.151,E2 -22632.151} C_VEL
LIN {X 0,Y 187.999,Z 558.792,A -85,B 0,C 180,E1 -22632.33,E2 -22632.33} C_VEL
LIN {X 0,Y 186.466,Z 558.451,A -85,B 0,C 180,E1 -22632.796,E2 -22632.796} C_VEL
LIN {X 0,Y 185.202,Z 557.001,A -85,B 0,C 180,E1 -22633.292,E2 -22633.292} C_VEL
LIN {X 0,Y 189.89,Z 570.57,A -85,B 0,C 180,E1 -22634.498,E2 -22634.498} C_VEL
LIN {X 0,Y 186.438,Z 632.053,A -85,B 0,C 180,E1 -22638.002,E2 -22638.002} C_VEL
LIN {X 0,Y 185.519,Z 645.175,A -85,B 0,C 180,E1 -22639.149,E2 -22639.149} C_VEL
LIN {X 0,Y 184.262,Z 657.697,A -85,B 0,C 180,E1 -22640.646,E2 -22640.646} C_VEL
LIN {X 0,Y 182.709,Z 670.767,A -85,B 0,C 180,E1 -22642.711,E2 -22642.711} C_VEL
LIN {X 0,Y 181.261,Z 682.671,A -85,B 0,C 180,E1 -22645.116,E2 -22645.116} C_VEL
LIN {X 0,Y 179.632,Z 694.443,A -85,B 0,C 180,E1 -22648.117,E2 -22648.117} C_VEL
LIN {X 0,Y 178.376,Z 704.021,A -85,B 0,C 180,E1 -22651.185,E2 -22651.185} C_VEL
LIN {X 0,Y 177.418,Z 712.937,A -85,B 0,C 180,E1 -22654.721,E2 -22654.721} C_VEL
LIN {X 0,Y 176.672,Z 720.299,A -85,B 0,C 180,E1 -22658.409,E2 -22658.409} C_VEL
LIN {X 0,Y 176.385,Z 726.385,A -85,B 0,C 180,E1 -22662.341,E2 -22662.341} C_VEL
LIN {X 0,Y 176.617,Z 730.935,A -85,B 0,C 180,E1 -22666.186,E2 -22666.186} C_VEL
LIN {X 0,Y 177.08,Z 733.101,A -85,B 0,C 180,E1 -22668.554,E2 -22668.554} C_VEL
LIN {X 0,Y 177.836,Z 734.924,A -85,B 0,C 180,E1 -22671.101,E2 -22671.101} C_VEL
LIN {X 0,Y 179.823,Z 736.929,A -85,B 0,C 180,E1 -22675.516,E2 -22675.516} C_VEL
LIN {X 0,Y 182.726,Z 737.368,A -85,B 0,C 180,E1 -22679.727,E2 -22679.727} C_VEL
LIN {X 0,Y 184.83,Z 736.969,A -85,B 0,C 180,E1 -22682.179,E2 -22682.179} C_VEL
LIN {X 0,Y 187.037,Z 736.186,A -85,B 0,C 180,E1 -22684.309,E2 -22684.309} C_VEL
LIN {X 0,Y 191.622,Z 733.682,A -85,B 0,C 180,E1 -22688.012,E2 -22688.012} C_VEL
LIN {X 0,Y 196.576,Z 730.031,A -85,B 0,C 180,E1 -22691.34,E2 -22691.34} C_VEL
LIN {X 0,Y 201.626,Z 725.682,A -85,B 0,C 180,E1 -22694.122,E2 -22694.122} C_VEL
LIN {X 0,Y 207.138,Z 720.128,A -85,B 0,C 180,E1 -22696.762,E2 -22696.762} C_VEL
LIN {X 0,Y 214.065,Z 711.955,A -85,B 0,C 180,E1 -22699.665,E2 -22699.665} C_VEL
LIN {X 0,Y 219.615,Z 704.458,A -85,B 0,C 180,E1 -22701.671,E2 -22701.671} C_VEL
LIN {X 0,Y 226.155,Z 694.112,A -85,B 0,C 180,E1 -22703.827,E2 -22703.827} C_VEL
LIN {X 0,Y 232.1,Z 683.132,A -85,B 0,C 180,E1 -22705.562,E2 -22705.562} C_VEL
LIN {X 0,Y 237.131,Z 671.928,A -85,B 0,C 180,E1 -22706.949,E2 -22706.949} C_VEL
LIN {X 0,Y 241.797,Z 658.873,A -85,B 0,C 180,E1 -22708.186,E2 -22708.186} C_VEL
LIN {X 0,Y 245.482,Z 645.71,A -85,B 0,C 180,E1 -22709.124,E2 -22709.124} C_VEL
LIN {X 0,Y 247.077,Z 638.442,A -85,B 0,C 180,E1 -22709.491,E2 -22709.491} C_VEL
LIN {X 0,Y 247.538,Z 635.353,A -85,B 0,C 180,E1 -22709.795,E2 -22709.795} C_VEL
LIN {X 0,Y 247.707,Z 631.789,A -85,B 0,C 180,E1 -22710.544,E2 -22710.544} C_VEL
LIN {X 0,Y 247.507,Z 628.868,A -85,B 0,C 180,E1 -22711.675,E2 -22711.675} C_VEL
LIN {X 0,Y 247.135,Z 627.172,A -85,B 0,C 180,E1 -22712.964,E2 -22712.964} C_VEL
LIN {X 0,Y 246.911,Z 626.864,A -85,B 0,C 180,E1 -22713.635,E2 -22713.635} C_VEL
LIN {X 0,Y 246.374,Z 627.135,A -85,B 0,C 180,E1 -22716.062,E2 -22716.062} C_VEL
LIN {X 0,Y 246.303,Z 628.489,A -85,B 0,C 180,E1 -22717.846,E2 -22717.846} C_VEL
LIN {X 0,Y 246.534,Z 632.459,A -85,B 0,C 180,E1 -22720.481,E2 -22720.481} C_VEL
LIN {X 0,Y 246.692,Z 634.708,A -85,B 0,C 180,E1 -22721.519,E2 -22721.519} C_VEL
LIN {X 0,Y 242.873,Z 653.036,A -85,B 0,C 180,E1 -22722.296,E2 -22722.296} C_VEL
LIN {X 0,Y 238.987,Z 666.125,A -85,B 0,C 180,E1 -22722.975,E2 -22722.975} C_VEL
LIN {X 0,Y 233.883,Z 679.354,A -85,B 0,C 180,E1 -22723.849,E2 -22723.849} C_VEL
LIN {X 0,Y 228.339,Z 691.171,A -85,B 0,C 180,E1 -22724.936,E2 -22724.936} C_VEL
LIN {X 0,Y 221.633,Z 703.32,A -85,B 0,C 180,E1 -22726.395,E2 -22726.395} C_VEL
LIN {X 0,Y 215.267,Z 713.28,A -85,B 0,C 180,E1 -22727.99,E2 -22727.99} C_VEL
LIN {X 0,Y 208.055,Z 723.148,A -85,B 0,C 180,E1 -22730.074,E2 -22730.074} C_VEL
LIN {X 0,Y 201.408,Z 731.354,A -85,B 0,C 180,E1 -22732.364,E2 -22732.364} C_VEL
LIN {X 0,Y 194.249,Z 739.201,A -85,B 0,C 180,E1 -22735.262,E2 -22735.262} C_VEL
LIN {X 0,Y 187.889,Z 745.504,A -85,B 0,C 180,E1 -22738.422,E2 -22738.422} C_VEL
LIN {X 0,Y 181.727,Z 751.005,A -85,B 0,C 180,E1 -22742.35,E2 -22742.35} C_VEL
LIN {X 0,Y 176.797,Z 754.993,A -85,B 0,C 180,E1 -22746.577,E2 -22746.577} C_VEL
LIN {X 0,Y 174.704,Z 756.446,A -85,B 0,C 180,E1 -22748.774,E2 -22748.774} C_VEL
LIN {X 0,Y 172.488,Z 762.609,A -85,B 0,C 180,E1 -22752.207,E2 -22752.207} C_VEL
LIN {X 0,Y 170.713,Z 767.484,A -85,B 0,C 180,E1 -22755.7,E2 -22755.7} C_VEL
LIN {X 0,Y 169.676,Z 771.228,A -85,B 0,C 180,E1 -22759.258,E2 -22759.258} C_VEL
LIN {X 0,Y 169.098,Z 773.937,A -85,B 0,C 180,E1 -22762.838,E2 -22762.838} C_VEL
LIN {X 0,Y 168.898,Z 775.885,A -85,B 0,C 180,E1 -22767.029,E2 -22767.029} C_VEL
LIN {X 0,Y 169.001,Z 776.499,A -85,B 0,C 180,E1 -22770,E2 -22770} C_VEL
LIN {X 0,Y 168.91,Z 776.47,A -85,B 0,C 180,E1 -22773.043,E2 -22773.043} C_VEL
LIN {X 0,Y 169.099,Z 775.374,A -85,B 0,C 180,E1 -22777.162,E2 -22777.162} C_VEL
LIN {X 0,Y 170.054,Z 772.537,A -85,B 0,C 180,E1 -22781.925,E2 -22781.925} C_VEL
LIN {X 0,Y 171.305,Z 769.28,A -85,B 0,C 180,E1 -22785.466,E2 -22785.466} C_VEL
LIN {X 0,Y 173.344,Z 764.952,A -85,B 0,C 180,E1 -22788.926,E2 -22788.926} C_VEL
LIN {X 0,Y 175.924,Z 759.422,A -85,B 0,C 180,E1 -22792.303,E2 -22792.303} C_VEL
LIN {X 0,Y 179,Z 752.507,A -85,B 0,C 180,E1 -22795.587,E2 -22795.587} C_VEL
LIN {X 0,Y 182.632,Z 743.835,A -85,B 0,C 180,E1 -22798.751,E2 -22798.751} C_VEL
LIN {X 0,Y 186.591,Z 733.981,A -85,B 0,C 180,E1 -22801.506,E2 -22801.506} C_VEL
LIN {X 0,Y 190.142,Z 723.912,A -85,B 0,C 180,E1 -22803.67,E2 -22803.67} C_VEL
LIN {X 0,Y 193.484,Z 712.755,A -85,B 0,C 180,E1 -22805.532,E2 -22805.532} C_VEL
LIN {X 0,Y 196.459,Z 701.2,A -85,B 0,C 180,E1 -22806.972,E2 -22806.972} C_VEL
LIN {X 0,Y 198.913,Z 688.562,A -85,B 0,C 180,E1 -22808.111,E2 -22808.111} C_VEL
LIN {X 0,Y 200.722,Z 675.258,A -85,B 0,C 180,E1 -22808.906,E2 -22808.906} C_VEL
LIN {X 0,Y 202.437,Z 647.276,A -85,B 0,C 180,E1 -22809.876,E2 -22809.876} C_VEL
LIN {X 0,Y 203.838,Z 620.415,A -85,B 0,C 180,E1 -22810.764,E2 -22810.764} C_VEL
LIN {X 0,Y 202.051,Z 598.05,A -85,B 0,C 180,E1 -22812.272,E2 -22812.272} C_VEL
LIN {X 0,Y 201.425,Z 593.776,A -85,B 0,C 180,E1 -22812.644,E2 -22812.644} C_VEL
LIN {X 0,Y 196.708,Z 580.555,A -85,B 0,C 180,E1 -22814.633,E2 -22814.633} C_VEL
LIN {X 0,Y 190.377,Z 570.258,A -85,B 0,C 180,E1 -22817.172,E2 -22817.172} C_VEL
LIN {X 0,Y 184.097,Z 560.886,A -85,B 0,C 180,E1 -22819.957,E2 -22819.957} C_VEL
LIN {X 0,Y 181.317,Z 556.781,A -85,B 0,C 180,E1 -22821.376,E2 -22821.376} C_VEL
LIN {X 0,Y 178.831,Z 551.95,A -85,B 0,C 180,E1 -22823.879,E2 -22823.879} C_VEL
LIN {X 0,Y 175.303,Z 545.627,A -85,B 0,C 180,E1 -22827.726,E2 -22827.726} C_VEL
LIN {X 0,Y 173.527,Z 542.237,A -85,B 0,C 180,E1 -22830.025,E2 -22830.025} C_VEL
LIN {X 0,Y 171.954,Z 539.999,A -85,B 0,C 180,E1 -22831.965,E2 -22831.965} C_VEL
LIN {X 0,Y 171.411,Z 538.124,A -85,B 0,C 180,E1 -22833.192,E2 -22833.192} C_VEL
LIN {X 0,Y 171.449,Z 538.111,A -85,B 0,C 180,E1 -22838.351,E2 -22838.351} C_VEL
LIN {X 0,Y 171.574,Z 538.096,A -85,B 0,C 180,E1 -22840.872,E2 -22840.872} C_VEL
LIN {X 0,Y 171.588,Z 538.088,A -85,B 0,C 180,E1 -22845.774,E2 -22845.774} C_VEL
LIN {X 0,Y 171.869,Z 538.038,A -85,B 0,C 180,E1 -22850.587,E2 -22850.587} C_VEL
LIN {X 0,Y 171.82,Z 538.08,A -85,B 0,C 180,E1 -22855.308,E2 -22855.308} C_VEL
LIN {X 0,Y 172.329,Z 537.976,A -85,B 0,C 180,E1 -22860.001,E2 -22860.001} C_VEL
LIN {X 0,Y 171.815,Z 538.082,A -85,B 0,C 180,E1 -22864.693,E2 -22864.693} C_VEL
LIN {X 0,Y 171.845,Z 538.042,A -85,B 0,C 180,E1 -22869.416,E2 -22869.416} C_VEL
LIN {X 0,Y 171.573,Z 538.09,A -85,B 0,C 180,E1 -22874.228,E2 -22874.228} C_VEL
LIN {X 0,Y 171.555,Z 538.114,A -85,B 0,C 180,E1 -22879.575,E2 -22879.575} C_VEL
LIN {X 0,Y 171.455,Z 538.104,A -85,B 0,C 180,E1 -22883.878,E2 -22883.878} C_VEL
LIN {X 0,Y 172.702,Z 541.319,A -85,B 0,C 180,E1 -22886.593,E2 -22886.593} C_VEL
LIN {X 0,Y 173.52,Z 542.539,A -85,B 0,C 180,E1 -22887.761,E2 -22887.761} C_VEL
LIN {X 0,Y 176.359,Z 548.953,A -85,B 0,C 180,E1 -22892.549,E2 -22892.549} C_VEL
LIN {X 0,Y 178.294,Z 553.436,A -85,B 0,C 180,E1 -22895.378,E2 -22895.378} C_VEL
LIN {X 0,Y 182.975,Z 560.346,A -85,B 0,C 180,E1 -22897.755,E2 -22897.755} C_VEL
LIN {X 0,Y 188.475,Z 568.757,A -85,B 0,C 180,E1 -22900.276,E2 -22900.276} C_VEL
LIN {X 0,Y 194.643,Z 579.518,A -85,B 0,C 180,E1 -22902.872,E2 -22902.872} C_VEL
LIN {X 0,Y 200.24,Z 590.843,A -85,B 0,C 180,E1 -22905.073,E2 -22905.073} C_VEL
LIN {X 0,Y 205.339,Z 603.036,A -85,B 0,C 180,E1 -22906.996,E2 -22906.996} C_VEL
LIN {X 0,Y 201.624,Z 665.301,A -85,B 0,C 180,E1 -22909.025,E2 -22909.025} C_VEL
LIN {X 0,Y 200.024,Z 678.327,A -85,B 0,C 180,E1 -22909.789,E2 -22909.789} C_VEL
LIN {X 0,Y 197.835,Z 690.807,A -85,B 0,C 180,E1 -22910.91,E2 -22910.91} C_VEL
LIN {X 0,Y 194.974,Z 703.299,A -85,B 0,C 180,E1 -22912.469,E2 -22912.469} C_VEL
LIN {X 0,Y 191.73,Z 714.823,A -85,B 0,C 180,E1 -22914.416,E2 -22914.416} C_VEL
LIN {X 0,Y 188.197,Z 724.948,A -85,B 0,C 180,E1 -22916.577,E2 -22916.577} C_VEL
LIN {X 0,Y 184.597,Z 734.05,A -85,B 0,C 180,E1 -22919.072,E2 -22919.072} C_VEL
LIN {X 0,Y 180.774,Z 742.849,A -85,B 0,C 180,E1 -22922.192,E2 -22922.192} C_VEL
LIN {X 0,Y 177.884,Z 749.166,A -85,B 0,C 180,E1 -22925.057,E2 -22925.057} C_VEL
LIN {X 0,Y 174.935,Z 755.557,A -85,B 0,C 180,E1 -22928.804,E2 -22928.804} C_VEL
LIN {X 0,Y 172.668,Z 759.958,A -85,B 0,C 180,E1 -22932.226,E2 -22932.226} C_VEL
LIN {X 0,Y 171.011,Z 763.275,A -85,B 0,C 180,E1 -22935.725,E2 -22935.725} C_VEL
LIN {X 0,Y 170.224,Z 764.913,A -85,B 0,C 180,E1 -22938.087,E2 -22938.087} C_VEL
LIN {X 0,Y 169.214,Z 767.001,A -85,B 0,C 180,E1 -22942.843,E2 -22942.843} C_VEL
LIN {X 0,Y 168.932,Z 767.488,A -85,B 0,C 180,E1 -22946.835,E2 -22946.835} C_VEL
LIN {X 0,Y 169.002,Z 767.079,A -85,B 0,C 180,E1 -22950,E2 -22950} C_VEL
LIN {X 0,Y 169.152,Z 766.334,A -85,B 0,C 180,E1 -22952.381,E2 -22952.381} C_VEL
LIN {X 0,Y 169.51,Z 765.151,A -85,B 0,C 180,E1 -22954.756,E2 -22954.756} C_VEL
LIN {X 0,Y 169.987,Z 763.572,A -85,B 0,C 180,E1 -22957.125,E2 -22957.125} C_VEL
LIN {X 0,Y 171.008,Z 760.392,A -85,B 0,C 180,E1 -22960.657,E2 -22960.657} C_VEL
LIN {X 0,Y 172.605,Z 756.147,A -85,B 0,C 180,E1 -22964.14,E2 -22964.14} C_VEL
LIN {X 0,Y 174.744,Z 750.719,A -85,B 0,C 180,E1 -22967.556,E2 -22967.556} C_VEL
LIN {X 0,Y 177.412,Z 743.924,A -85,B 0,C 180,E1 -22970.886,E2 -22970.886} C_VEL
LIN {X 0,Y 180.594,Z 735.384,A -85,B 0,C 180,E1 -22974.117,E2 -22974.117} C_VEL
LIN {X 0,Y 183.565,Z 726.641,A -85,B 0,C 180,E1 -22976.734,E2 -22976.734} C_VEL
LIN {X 0,Y 186.636,Z 717.042,A -85,B 0,C 180,E1 -22979,E2 -22979} C_VEL
LIN {X 0,Y 189.588,Z 706.439,A -85,B 0,C 180,E1 -22980.953,E2 -22980.953} C_VEL
LIN {X 0,Y 191.944,Z 695.948,A -85,B 0,C 180,E1 -22982.474,E2 -22982.474} C_VEL
LIN {X 0,Y 194.075,Z 683.656,A -85,B 0,C 180,E1 -22983.832,E2 -22983.832} C_VEL
LIN {X 0,Y 195.678,Z 671.581,A -85,B 0,C 180,E1 -22984.761,E2 -22984.761} C_VEL
LIN {X 0,Y 196.805,Z 657.573,A -85,B 0,C 180,E1 -22985.411,E2 -22985.411} C_VEL
LIN {X 0,Y 199.935,Z 599.611,A -85,B 0,C 180,E1 -22987.313,E2 -22987.313} C_VEL
LIN {X 0,Y 199.262,Z 595.28,A -85,B 0,C 180,E1 -22987.663,E2 -22987.663} C_VEL
LIN {X 0,Y 193.996,Z 582.709,A -85,B 0,C 180,E1 -22989.522,E2 -22989.522} C_VEL
LIN {X 0,Y 187.644,Z 569.8,A -85,B 0,C 180,E1 -22991.866,E2 -22991.866} C_VEL
LIN {X 0,Y 187.316,Z 569.253,A -85,B 0,C 180,E1 -22991.987,E2 -22991.987} C_VEL
LIN {X 0,Y 186.202,Z 569.508,A -85,B 0,C 180,E1 -22992.295,E2 -22992.295} C_VEL
LIN {X 0,Y 185.286,Z 570.227,A -85,B 0,C 180,E1 -22992.526,E2 -22992.526} C_VEL
LIN {X 0,Y 182.752,Z 569.868,A -85,B 0,C 180,E1 -22993.307,E2 -22993.307} C_VEL
LIN {X 0,Y 181.791,Z 568.504,A -85,B 0,C 180,E1 -22993.679,E2 -22993.679} C_VEL
LIN {X 0,Y 182.95,Z 571.921,A -85,B 0,C 180,E1 -22994.028,E2 -22994.028} C_VEL
LIN {X 0,Y 179.422,Z 632.669,A -85,B 0,C 180,E1 -22997.681,E2 -22997.681} C_VEL
LIN {X 0,Y 178.429,Z 645.972,A -85,B 0,C 180,E1 -22998.906,E2 -22998.906} C_VEL
LIN {X 0,Y 177.064,Z 659.164,A -85,B 0,C 180,E1 -23000.574,E2 -23000.574} C_VEL
LIN {X 0,Y 175.494,Z 672.061,A -85,B 0,C 180,E1 -23002.719,E2 -23002.719} C_VEL
LIN {X 0,Y 174.014,Z 683.78,A -85,B 0,C 180,E1 -23005.217,E2 -23005.217} C_VEL
LIN {X 0,Y 172.516,Z 694.372,A -85,B 0,C 180,E1 -23008.021,E2 -23008.021} C_VEL
LIN {X 0,Y 171.264,Z 703.991,A -85,B 0,C 180,E1 -23011.172,E2 -23011.172} C_VEL
LIN {X 0,Y 170.397,Z 712.074,A -85,B 0,C 180,E1 -23014.455,E2 -23014.455} C_VEL
LIN {X 0,Y 169.621,Z 719.354,A -85,B 0,C 180,E1 -23018.105,E2 -23018.105} C_VEL
LIN {X 0,Y 169.322,Z 725.274,A -85,B 0,C 180,E1 -23021.803,E2 -23021.803} C_VEL
LIN {X 0,Y 169.445,Z 730.024,A -85,B 0,C 180,E1 -23025.589,E2 -23025.589} C_VEL
LIN {X 0,Y 169.871,Z 732.466,A -85,B 0,C 180,E1 -23028.061,E2 -23028.061} C_VEL
LIN {X 0,Y 170.708,Z 734.901,A -85,B 0,C 180,E1 -23031.134,E2 -23031.134} C_VEL
LIN {X 0,Y 172.52,Z 737.108,A -85,B 0,C 180,E1 -23035.326,E2 -23035.326} C_VEL
LIN {X 0,Y 175.656,Z 738.098,A -85,B 0,C 180,E1 -23039.999,E2 -23039.999} C_VEL
LIN {X 0,Y 177.597,Z 738.01,A -85,B 0,C 180,E1 -23042.267,E2 -23042.267} C_VEL
LIN {X 0,Y 179.835,Z 737.484,A -85,B 0,C 180,E1 -23044.482,E2 -23044.482} C_VEL
LIN {X 0,Y 184.755,Z 735.375,A -85,B 0,C 180,E1 -23048.504,E2 -23048.504} C_VEL
LIN {X 0,Y 189.635,Z 732.427,A -85,B 0,C 180,E1 -23051.761,E2 -23051.761} C_VEL
LIN {X 0,Y 194.793,Z 728.586,A -85,B 0,C 180,E1 -23054.628,E2 -23054.628} C_VEL
LIN {X 0,Y 200.457,Z 723.622,A -85,B 0,C 180,E1 -23057.338,E2 -23057.338} C_VEL
LIN {X 0,Y 206.557,Z 717.46,A -85,B 0,C 180,E1 -23059.892,E2 -23059.892} C_VEL
LIN {X 0,Y 213.048,Z 709.799,A -85,B 0,C 180,E1 -23062.266,E2 -23062.266} C_VEL
LIN {X 0,Y 220.089,Z 700.233,A -85,B 0,C 180,E1 -23064.527,E2 -23064.527} C_VEL
LIN {X 0,Y 226.302,Z 690.255,A -85,B 0,C 180,E1 -23066.316,E2 -23066.316} C_VEL
LIN {X 0,Y 232.302,Z 678.755,A -85,B 0,C 180,E1 -23067.923,E2 -23067.923} C_VEL
LIN {X 0,Y 236.916,Z 668.246,A -85,B 0,C 180,E1 -23069.062,E2 -23069.062} C_VEL
LIN {X 0,Y 241.489,Z 655.04,A -85,B 0,C 180,E1 -23070.172,E2 -23070.172} C_VEL
LIN {X 0,Y 244.837,Z 642.262,A -85,B 0,C 180,E1 -23070.954,E2 -23070.954} C_VEL
LIN {X 0,Y 247.735,Z 627.856,A -85,B 0,C 180,E1 -23071.616,E2 -23071.616} C_VEL
LIN {X 0,Y 246.911,Z 626.864,A -85,B 0,C 180,E1 -23073.635,E2 -23073.635} C_VEL
LIN {X 0,Y 246.54,Z 627.442,A -85,B 0,C 180,E1 -23074.527,E2 -23074.527} C_VEL
LIN {X 0,Y 245.868,Z 629.72,A -85,B 0,C 180,E1 -23075.629,E2 -23075.629} C_VEL
LIN {X 0,Y 244.797,Z 634.938,A -85,B 0,C 180,E1 -23077.498,E2 -23077.498} C_VEL
LIN {X 0,Y 244.659,Z 636.088,A -85,B 0,C 180,E1 -23078.081,E2 -23078.081} C_VEL
LIN {X 0,Y 244.762,Z 639.042,A -85,B 0,C 180,E1 -23079.975,E2 -23079.975} C_VEL
LIN {X 0,Y 244.57,Z 640.225,A -85,B 0,C 180,E1 -23080.104,E2 -23080.104} C_VEL
LIN {X 0,Y 241.064,Z 654.869,A -85,B 0,C 180,E1 -23080.713,E2 -23080.713} C_VEL
LIN {X 0,Y 236.587,Z 668.414,A -85,B 0,C 180,E1 -23081.424,E2 -23081.424} C_VEL
LIN {X 0,Y 231.092,Z 681.472,A -85,B 0,C 180,E1 -23082.306,E2 -23082.306} C_VEL
LIN {X 0,Y 225.413,Z 692.735,A -85,B 0,C 180,E1 -23083.35,E2 -23083.35} C_VEL
LIN {X 0,Y 218.749,Z 703.921,A -85,B 0,C 180,E1 -23084.699,E2 -23084.699} C_VEL
LIN {X 0,Y 210.187,Z 716.186,A -85,B 0,C 180,E1 -23086.73,E2 -23086.73} C_VEL
LIN {X 0,Y 202.79,Z 725.401,A -85,B 0,C 180,E1 -23088.818,E2 -23088.818} C_VEL
LIN {X 0,Y 193.747,Z 735.299,A -85,B 0,C 180,E1 -23091.928,E2 -23091.928} C_VEL
LIN {X 0,Y 187.536,Z 741.297,A -85,B 0,C 180,E1 -23094.489,E2 -23094.489} C_VEL
LIN {X 0,Y 180.204,Z 747.622,A -85,B 0,C 180,E1 -23098.231,E2 -23098.231} C_VEL
LIN {X 0,Y 175.468,Z 751.32,A -85,B 0,C 180,E1 -23101.274,E2 -23101.274} C_VEL
LIN {X 0,Y 170.283,Z 754.885,A -85,B 0,C 180,E1 -23105.625,E2 -23105.625} C_VEL
LIN {X 0,Y 168.113,Z 756.187,A -85,B 0,C 180,E1 -23107.899,E2 -23107.899} C_VEL
LIN {X 0,Y 165.702,Z 762.36,A -85,B 0,C 180,E1 -23111.452,E2 -23111.452} C_VEL
LIN {X 0,Y 163.794,Z 767.247,A -85,B 0,C 180,E1 -23115.082,E2 -23115.082} C_VEL
LIN {X 0,Y 162.691,Z 771.003,A -85,B 0,C 180,E1 -23118.791,E2 -23118.791} C_VEL
LIN {X 0,Y 162.022,Z 773.722,A -85,B 0,C 180,E1 -23122.523,E2 -23122.523} C_VEL
LIN {X 0,Y 161.832,Z 775.789,A -85,B 0,C 180,E1 -23127.231,E2 -23127.231} C_VEL
LIN {X 0,Y 161.913,Z 776.305,A -85,B 0,C 180,E1 -23130,E2 -23130} C_VEL
LIN {X 0,Y 161.828,Z 776.312,A -85,B 0,C 180,E1 -23132.741,E2 -23132.741} C_VEL
LIN {X 0,Y 162.026,Z 775.199,A -85,B 0,C 180,E1 -23137.477,E2 -23137.477} C_VEL
LIN {X 0,Y 163.097,Z 772.375,A -85,B 0,C 180,E1 -23142.442,E2 -23142.442} C_VEL
LIN {X 0,Y 164.443,Z 769.129,A -85,B 0,C 180,E1 -23146.128,E2 -23146.128} C_VEL
LIN {X 0,Y 166.631,Z 764.814,A -85,B 0,C 180,E1 -23149.719,E2 -23149.719} C_VEL
LIN {X 0,Y 169.372,Z 759.299,A -85,B 0,C 180,E1 -23153.215,E2 -23153.215} C_VEL
LIN {X 0,Y 172.585,Z 752.403,A -85,B 0,C 180,E1 -23156.611,E2 -23156.611} C_VEL
LIN {X 0,Y 176.432,Z 743.754,A -85,B 0,C 180,E1 -23159.862,E2 -23159.862} C_VEL
LIN {X 0,Y 180.168,Z 734.89,A -85,B 0,C 180,E1 -23162.435,E2 -23162.435} C_VEL
LIN {X 0,Y 183.861,Z 725.142,A -85,B 0,C 180,E1 -23164.651,E2 -23164.651} C_VEL
LIN {X 0,Y 187.333,Z 714.337,A -85,B 0,C 180,E1 -23166.552,E2 -23166.552} C_VEL
LIN {X 0,Y 190.597,Z 702.259,A -85,B 0,C 180,E1 -23168.142,E2 -23168.142} C_VEL
LIN {X 0,Y 193.256,Z 689.531,A -85,B 0,C 180,E1 -23169.355,E2 -23169.355} C_VEL
LIN {X 0,Y 195.142,Z 676.777,A -85,B 0,C 180,E1 -23170.156,E2 -23170.156} C_VEL
LIN {X 0,Y 196.309,Z 660.726,A -85,B 0,C 180,E1 -23170.787,E2 -23170.787} C_VEL
LIN {X 0,Y 198.557,Z 621.319,A -85,B 0,C 180,E1 -23172.089,E2 -23172.089} C_VEL
LIN {X 0,Y 196.997,Z 600.292,A -85,B 0,C 180,E1 -23173.553,E2 -23173.553} C_VEL
LIN {X 0,Y 196.35,Z 596.101,A -85,B 0,C 180,E1 -23173.949,E2 -23173.949} C_VEL
LIN {X 0,Y 192.342,Z 584.79,A -85,B 0,C 180,E1 -23175.747,E2 -23175.747} C_VEL
LIN {X 0,Y 186.421,Z 574.981,A -85,B 0,C 180,E1 -23178.27,E2 -23178.27} C_VEL
LIN {X 0,Y 180.9,Z 566.533,A -85,B 0,C 180,E1 -23180.862,E2 -23180.862} C_VEL
LIN {X 0,Y 175.911,Z 559.524,A -85,B 0,C 180,E1 -23183.45,E2 -23183.45} C_VEL
LIN {X 0,Y 173.716,Z 556.354,A -85,B 0,C 180,E1 -23184.795,E2 -23184.795} C_VEL
LIN {X 0,Y 171.253,Z 551.558,A -85,B 0,C 180,E1 -23187.758,E2 -23187.758} C_VEL
LIN {X 0,Y 169.439,Z 548.091,A -85,B 0,C 180,E1 -23190.15,E2 -23190.15} C_VEL
LIN {X 0,Y 167.591,Z 545.339,A -85,B 0,C 180,E1 -23192.53,E2 -23192.53} C_VEL
LIN {X 0,Y 167.09,Z 543.712,A -85,B 0,C 180,E1 -23193.671,E2 -23193.671} C_VEL
LIN {X 0,Y 165.253,Z 541.565,A -85,B 0,C 180,E1 -23196.17,E2 -23196.17} C_VEL
LIN {X 0,Y 164.403,Z 538.99,A -85,B 0,C 180,E1 -23198.529,E2 -23198.529} C_VEL
LIN {X 0,Y 164.479,Z 538.959,A -85,B 0,C 180,E1 -23202.597,E2 -23202.597} C_VEL
LIN {X 0,Y 164.747,Z 538.945,A -85,B 0,C 180,E1 -23208.855,E2 -23208.855} C_VEL
LIN {X 0,Y 164.843,Z 538.912,A -85,B 0,C 180,E1 -23212.652,E2 -23212.652} C_VEL
LIN {X 0,Y 165.047,Z 538.902,A -85,B 0,C 180,E1 -23217.56,E2 -23217.56} C_VEL
LIN {X 0,Y 165.292,Z 538.852,A -85,B 0,C 180,E1 -23220.001,E2 -23220.001} C_VEL
LIN {X 0,Y 164.764,Z 538.958,A -85,B 0,C 180,E1 -23224.894,E2 -23224.894} C_VEL
LIN {X 0,Y 164.828,Z 538.915,A -85,B 0,C 180,E1 -23227.35,E2 -23227.35} C_VEL
LIN {X 0,Y 164.7,Z 538.95,A -85,B 0,C 180,E1 -23231.061,E2 -23231.061} C_VEL
LIN {X 0,Y 164.492,Z 538.962,A -85,B 0,C 180,E1 -23237.403,E2 -23237.403} C_VEL
LIN {X 0,Y 164.559,Z 539.091,A -85,B 0,C 180,E1 -23238.923,E2 -23238.923} C_VEL
LIN {X 0,Y 164.879,Z 540.625,A -85,B 0,C 180,E1 -23240.327,E2 -23240.327} C_VEL
LIN {X 0,Y 166.629,Z 543.377,A -85,B 0,C 180,E1 -23243.622,E2 -23243.622} C_VEL
LIN {X 0,Y 168.495,Z 547.415,A -85,B 0,C 180,E1 -23247.311,E2 -23247.311} C_VEL
LIN {X 0,Y 171.268,Z 553.693,A -85,B 0,C 180,E1 -23252.067,E2 -23252.067} C_VEL
LIN {X 0,Y 176.606,Z 561.203,A -85,B 0,C 180,E1 -23255.155,E2 -23255.155} C_VEL
LIN {X 0,Y 179.903,Z 566.157,A -85,B 0,C 180,E1 -23256.889,E2 -23256.889} C_VEL
LIN {X 0,Y 185.104,Z 574.419,A -85,B 0,C 180,E1 -23259.404,E2 -23259.404} C_VEL
LIN {X 0,Y 190.799,Z 584.608,A -85,B 0,C 180,E1 -23261.933,E2 -23261.933} C_VEL
LIN {X 0,Y 196.385,Z 596.348,A -85,B 0,C 180,E1 -23264.257,E2 -23264.257} C_VEL
LIN {X 0,Y 199.978,Z 605.188,A -85,B 0,C 180,E1 -23265.7,E2 -23265.7} C_VEL
LIN {X 0,Y 196.208,Z 665.977,A -85,B 0,C 180,E1 -23267.723,E2 -23267.723} C_VEL
LIN {X 0,Y 194.534,Z 678.782,A -85,B 0,C 180,E1 -23268.494,E2 -23268.494} C_VEL
LIN {X 0,Y 192.143,Z 691.743,A -85,B 0,C 180,E1 -23269.689,E2 -23269.689} C_VEL
LIN {X 0,Y 189.304,Z 703.496,A -85,B 0,C 180,E1 -23271.193,E2 -23271.193} C_VEL
LIN {X 0,Y 186.002,Z 714.821,A -85,B 0,C 180,E1 -23273.143,E2 -23273.143} C_VEL
LIN {X 0,Y 182.301,Z 724.98,A -85,B 0,C 180,E1 -23275.346,E2 -23275.346} C_VEL
LIN {X 0,Y 178.537,Z 734.12,A -85,B 0,C 180,E1 -23277.9,E2 -23277.9} C_VEL
LIN {X 0,Y 174.504,Z 742.94,A -85,B 0,C 180,E1 -23281.1,E2 -23281.1} C_VEL
LIN {X 0,Y 170.984,Z 750.246,A -85,B 0,C 180,E1 -23284.558,E2 -23284.558} C_VEL
LIN {X 0,Y 168.28,Z 755.688,A -85,B 0,C 180,E1 -23287.922,E2 -23287.922} C_VEL
LIN {X 0,Y 165.899,Z 760.104,A -85,B 0,C 180,E1 -23291.475,E2 -23291.475} C_VEL
LIN {X 0,Y 164.12,Z 763.434,A -85,B 0,C 180,E1 -23295.112,E2 -23295.112} C_VEL
LIN {X 0,Y 162.599,Z 766.325,A -85,B 0,C 180,E1 -23300.044,E2 -23300.044} C_VEL
LIN {X 0,Y 162.163,Z 767.18,A -85,B 0,C 180,E1 -23302.53,E2 -23302.53} C_VEL
LIN {X 0,Y 161.839,Z 767.649,A -85,B 0,C 180,E1 -23307.203,E2 -23307.203} C_VEL
LIN {X 0,Y 161.915,Z 767.279,A -85,B 0,C 180,E1 -23310,E2 -23310} C_VEL
LIN {X 0,Y 162.074,Z 766.543,A -85,B 0,C 180,E1 -23312.485,E2 -23312.485} C_VEL
LIN {X 0,Y 162.779,Z 764.273,A -85,B 0,C 180,E1 -23316.761,E2 -23316.761} C_VEL
LIN {X 0,Y 164.054,Z 760.626,A -85,B 0,C 180,E1 -23321.115,E2 -23321.115} C_VEL
LIN {X 0,Y 165.733,Z 756.394,A -85,B 0,C 180,E1 -23324.74,E2 -23324.74} C_VEL
LIN {X 0,Y 168.011,Z 750.979,A -85,B 0,C 180,E1 -23328.284,E2 -23328.284} C_VEL
LIN {X 0,Y 170.815,Z 744.203,A -85,B 0,C 180,E1 -23331.733,E2 -23331.733} C_VEL
LIN {X 0,Y 174.153,Z 735.685,A -85,B 0,C 180,E1 -23335.07,E2 -23335.07} C_VEL
LIN {X 0,Y 177.281,Z 726.962,A -85,B 0,C 180,E1 -23337.762,E2 -23337.762} C_VEL
LIN {X 0,Y 180.487,Z 717.387,A -85,B 0,C 180,E1 -23340.088,E2 -23340.088} C_VEL
LIN {X 0,Y 183.561,Z 706.835,A -85,B 0,C 180,E1 -23342.088,E2 -23342.088} C_VEL
LIN {X 0,Y 186.005,Z 696.393,A -85,B 0,C 180,E1 -23343.646,E2 -23343.646} C_VEL
LIN {X 0,Y 188.237,Z 684.173,A -85,B 0,C 180,E1 -23345.031,E2 -23345.031} C_VEL
LIN {X 0,Y 190.018,Z 671.306,A -85,B 0,C 180,E1 -23346.036,E2 -23346.036} C_VEL
LIN {X 0,Y 191.177,Z 657.038,A -85,B 0,C 180,E1 -23346.695,E2 -23346.695} C_VEL
LIN {X 0,Y 194.361,Z 599.868,A -85,B 0,C 180,E1 -23348.616,E2 -23348.616} C_VEL
LIN {X 0,Y 193.644,Z 597.261,A -85,B 0,C 180,E1 -23348.916,E2 -23348.916} C_VEL
LIN {X 0,Y 188.394,Z 584.718,A -85,B 0,C 180,E1 -23350.898,E2 -23350.898} C_VEL
LIN {X 0,Y 185.137,Z 577.941,A -85,B 0,C 180,E1 -23352.165,E2 -23352.165} C_VEL
LIN {X 0,Y 184.895,Z 577.904,A -85,B 0,C 180,E1 -23352.238,E2 -23352.238} C_VEL
LIN {X 0,Y 181.16,Z 589.057,A -85,B 0,C 180,E1 -23352.758,E2 -23352.758} C_VEL
LIN {X 0,Y 178.553,Z 594.373,A -85,B 0,C 180,E1 -23353.273,E2 -23353.273} C_VEL
LIN {X 0,Y 177.071,Z 596.124,A -85,B 0,C 180,E1 -23353.646,E2 -23353.646} C_VEL
LIN {X 0,Y 175.78,Z 595.946,A -85,B 0,C 180,E1 -23354.074,E2 -23354.074} C_VEL
LIN {X 0,Y 175.054,Z 593.613,A -85,B 0,C 180,E1 -23354.448,E2 -23354.448} C_VEL
LIN {X 0,Y 174.789,Z 591.347,A -85,B 0,C 180,E1 -23354.667,E2 -23354.667} C_VEL
LIN {X 0,Y 172.301,Z 634.232,A -85,B 0,C 180,E1 -23357.425,E2 -23357.425} C_VEL
LIN {X 0,Y 171.213,Z 647.949,A -85,B 0,C 180,E1 -23358.775,E2 -23358.775} C_VEL
LIN {X 0,Y 169.763,Z 661.675,A -85,B 0,C 180,E1 -23360.659,E2 -23360.659} C_VEL
LIN {X 0,Y 168.279,Z 673.071,A -85,B 0,C 180,E1 -23362.673,E2 -23362.673} C_VEL
LIN {X 0,Y 166.748,Z 684.82,A -85,B 0,C 180,E1 -23365.319,E2 -23365.319} C_VEL
LIN {X 0,Y 165.28,Z 695.297,A -85,B 0,C 180,E1 -23368.257,E2 -23368.257} C_VEL
LIN {X 0,Y 164.151,Z 703.903,A -85,B 0,C 180,E1 -23371.205,E2 -23371.205} C_VEL
LIN {X 0,Y 163.249,Z 712.234,A -85,B 0,C 180,E1 -23374.695,E2 -23374.695} C_VEL
LIN {X 0,Y 162.52,Z 719.481,A -85,B 0,C 180,E1 -23378.433,E2 -23378.433} C_VEL
LIN {X 0,Y 162.218,Z 725.626,A -85,B 0,C 180,E1 -23382.385,E2 -23382.385} C_VEL
LIN {X 0,Y 162.442,Z 730.294,A -85,B 0,C 180,E1 -23386.233,E2 -23386.233} C_VEL
LIN {X 0,Y 163.233,Z 733.89,A -85,B 0,C 180,E1 -23390.082,E2 -23390.082} C_VEL
LIN {X 0,Y 164.107,Z 735.727,A -85,B 0,C 180,E1 -23392.618,E2 -23392.618} C_VEL
LIN {X 0,Y 165.209,Z 737.109,A -85,B 0,C 180,E1 -23395.119,E2 -23395.119} C_VEL
LIN {X 0,Y 168.376,Z 738.673,A -85,B 0,C 180,E1 -23399.999,E2 -23399.999} C_VEL
LIN {X 0,Y 170.33,Z 738.848,A -85,B 0,C 180,E1 -23402.364,E2 -23402.364} C_VEL
LIN {X 0,Y 175.166,Z 737.959,A -85,B 0,C 180,E1 -23406.913,E2 -23406.913} C_VEL
LIN {X 0,Y 177.97,Z 736.948,A -85,B 0,C 180,E1 -23409.088,E2 -23409.088} C_VEL
LIN {X 0,Y 181.035,Z 735.515,A -85,B 0,C 180,E1 -23411.192,E2 -23411.192} C_VEL
LIN {X 0,Y 186.115,Z 732.521,A -85,B 0,C 180,E1 -23414.208,E2 -23414.208} C_VEL
LIN {X 0,Y 191.794,Z 728.515,A -85,B 0,C 180,E1 -23417.046,E2 -23417.046} C_VEL
LIN {X 0,Y 199.029,Z 722.326,A -85,B 0,C 180,E1 -23420.138,E2 -23420.138} C_VEL
LIN {X 0,Y 205.485,Z 715.857,A -85,B 0,C 180,E1 -23422.567,E2 -23422.567} C_VEL
LIN {X 0,Y 212.787,Z 707.434,A -85,B 0,C 180,E1 -23424.904,E2 -23424.904} C_VEL
LIN {X 0,Y 220.339,Z 697.016,A -85,B 0,C 180,E1 -23427.086,E2 -23427.086} C_VEL
LIN {X 0,Y 226.609,Z 686.874,A -85,B 0,C 180,E1 -23428.696,E2 -23428.696} C_VEL
LIN {X 0,Y 232.636,Z 675.019,A -85,B 0,C 180,E1 -23430.149,E2 -23430.149} C_VEL
LIN {X 0,Y 237.606,Z 663.119,A -85,B 0,C 180,E1 -23431.272,E2 -23431.272} C_VEL
LIN {X 0,Y 241.751,Z 650.48,A -85,B 0,C 180,E1 -23432.173,E2 -23432.173} C_VEL
LIN {X 0,Y 244.882,Z 637.531,A -85,B 0,C 180,E1 -23432.837,E2 -23432.837} C_VEL
LIN {X 0,Y 245.556,Z 634.041,A -85,B 0,C 180,E1 -23433.049,E2 -23433.049} C_VEL
LIN {X 0,Y 245.026,Z 633.788,A -85,B 0,C 180,E1 -23435.005,E2 -23435.005} C_VEL
LIN {X 0,Y 244.76,Z 634.739,A -85,B 0,C 180,E1 -23437.084,E2 -23437.084} C_VEL
LIN {X 0,Y 244.659,Z 636.088,A -85,B 0,C 180,E1 -23438.081,E2 -23438.081} C_VEL
LIN {X 0,Y 244.427,Z 637.758,A -85,B 0,C 180,E1 -23438.588,E2 -23438.588} C_VEL
LIN {X 0,Y 243.855,Z 640.835,A -85,B 0,C 180,E1 -23438.955,E2 -23438.955} C_VEL
LIN {X 0,Y 242.993,Z 644.645,A -85,B 0,C 180,E1 -23439.098,E2 -23439.098} C_VEL
LIN {X 0,Y 240.056,Z 654.941,A -85,B 0,C 180,E1 -23439.042,E2 -23439.042} C_VEL
LIN {X 0,Y 239.627,Z 656.341,A -85,B 0,C 180,E1 -23439.09,E2 -23439.09} C_VEL
LIN {X 0,Y 235.135,Z 669.143,A -85,B 0,C 180,E1 -23439.747,E2 -23439.747} C_VEL
LIN {X 0,Y 229.174,Z 682.439,A -85,B 0,C 180,E1 -23440.626,E2 -23440.626} C_VEL
LIN {X 0,Y 222.677,Z 694.329,A -85,B 0,C 180,E1 -23441.724,E2 -23441.724} C_VEL
LIN {X 0,Y 214.854,Z 706.448,A -85,B 0,C 180,E1 -23443.23,E2 -23443.23} C_VEL
LIN {X 0,Y 207.892,Z 715.746,A -85,B 0,C 180,E1 -23444.773,E2 -23444.773} C_VEL
LIN {X 0,Y 200.143,Z 724.795,A -85,B 0,C 180,E1 -23446.786,E2 -23446.786} C_VEL
LIN {X 0,Y 192.888,Z 732.385,A -85,B 0,C 180,E1 -23449.018,E2 -23449.018} C_VEL
LIN {X 0,Y 186.087,Z 738.679,A -85,B 0,C 180,E1 -23451.454,E2 -23451.454} C_VEL
LIN {X 0,Y 177.909,Z 745.461,A -85,B 0,C 180,E1 -23455.055,E2 -23455.055} C_VEL
LIN {X 0,Y 172.499,Z 749.387,A -85,B 0,C 180,E1 -23458.019,E2 -23458.019} C_VEL
LIN {X 0,Y 166.397,Z 753.354,A -85,B 0,C 180,E1 -23462.316,E2 -23462.316} C_VEL
LIN {X 0,Y 161.566,Z 755.926,A -85,B 0,C 180,E1 -23466.953,E2 -23466.953} C_VEL
LIN {X 0,Y 158.959,Z 762.111,A -85,B 0,C 180,E1 -23470.635,E2 -23470.635} C_VEL
LIN {X 0,Y 156.901,Z 767.009,A -85,B 0,C 180,E1 -23474.41,E2 -23474.41} C_VEL
LIN {X 0,Y 155.681,Z 770.777,A -85,B 0,C 180,E1 -23478.279,E2 -23478.279} C_VEL
LIN {X 0,Y 154.965,Z 773.507,A -85,B 0,C 180,E1 -23482.18,E2 -23482.18} C_VEL
LIN {X 0,Y 154.759,Z 774.789,A -85,B 0,C 180,E1 -23484.789,E2 -23484.789} C_VEL
LIN {X 0,Y 154.738,Z 775.746,A -85,B 0,C 180,E1 -23487.719,E2 -23487.719} C_VEL
LIN {X 0,Y 154.812,Z 776.112,A -85,B 0,C 180,E1 -23490,E2 -23490} C_VEL
LIN {X 0,Y 154.738,Z 776.14,A -85,B 0,C 180,E1 -23492.603,E2 -23492.603} C_VEL
LIN {X 0,Y 154.76,Z 775.779,A -85,B 0,C 180,E1 -23495.211,E2 -23495.211} C_VEL
LIN {X 0,Y 154.972,Z 775.023,A -85,B 0,C 180,E1 -23497.819,E2 -23497.819} C_VEL
LIN {X 0,Y 155.433,Z 773.821,A -85,B 0,C 180,E1 -23500.42,E2 -23500.42} C_VEL
LIN {X 0,Y 156.541,Z 771.255,A -85,B 0,C 180,E1 -23504.295,E2 -23504.295} C_VEL
LIN {X 0,Y 158.298,Z 767.678,A -85,B 0,C 180,E1 -23508.106,E2 -23508.106} C_VEL
LIN {X 0,Y 160.846,Z 762.986,A -85,B 0,C 180,E1 -23511.801,E2 -23511.801} C_VEL
LIN {X 0,Y 163.962,Z 757.035,A -85,B 0,C 180,E1 -23515.38,E2 -23515.38} C_VEL
LIN {X 0,Y 167.507,Z 749.624,A -85,B 0,C 180,E1 -23518.848,E2 -23518.848} C_VEL
LIN {X 0,Y 171.066,Z 742.064,A -85,B 0,C 180,E1 -23521.588,E2 -23521.588} C_VEL
LIN {X 0,Y 175.054,Z 732.857,A -85,B 0,C 180,E1 -23524.198,E2 -23524.198} C_VEL
LIN {X 0,Y 178.947,Z 722.614,A -85,B 0,C 180,E1 -23526.442,E2 -23526.442} C_VEL
LIN {X 0,Y 182.633,Z 711.26,A -85,B 0,C 180,E1 -23528.353,E2 -23528.353} C_VEL
LIN {X 0,Y 185.817,Z 699.298,A -85,B 0,C 180,E1 -23529.836,E2 -23529.836} C_VEL
LIN {X 0,Y 188.464,Z 686.091,A -85,B 0,C 180,E1 -23531.001,E2 -23531.001} C_VEL
LIN {X 0,Y 190.229,Z 673.191,A -85,B 0,C 180,E1 -23531.735,E2 -23531.735} C_VEL
LIN {X 0,Y 193.389,Z 622.26,A -85,B 0,C 180,E1 -23533.483,E2 -23533.483} C_VEL
LIN {X 0,Y 191.902,Z 601.29,A -85,B 0,C 180,E1 -23535.011,E2 -23535.011} C_VEL
LIN {X 0,Y 191.394,Z 598.603,A -85,B 0,C 180,E1 -23535.311,E2 -23535.311} C_VEL
LIN {X 0,Y 188.188,Z 589.305,A -85,B 0,C 180,E1 -23536.851,E2 -23536.851} C_VEL
LIN {X 0,Y 182.76,Z 580.051,A -85,B 0,C 180,E1 -23539.309,E2 -23539.309} C_VEL
LIN {X 0,Y 177.155,Z 571.245,A -85,B 0,C 180,E1 -23542.113,E2 -23542.113} C_VEL
LIN {X 0,Y 172.499,Z 564.651,A -85,B 0,C 180,E1 -23544.689,E2 -23544.689} C_VEL
LIN {X 0,Y 166.584,Z 556.595,A -85,B 0,C 180,E1 -23548.439,E2 -23548.439} C_VEL
LIN {X 0,Y 165.181,Z 553.831,A -85,B 0,C 180,E1 -23550.407,E2 -23550.407} C_VEL
LIN {X 0,Y 162.558,Z 549.06,A -85,B 0,C 180,E1 -23554.384,E2 -23554.384} C_VEL
LIN {X 0,Y 160.435,Z 545.571,A -85,B 0,C 180,E1 -23558.14,E2 -23558.14} C_VEL
LIN {X 0,Y 159.899,Z 544.413,A -85,B 0,C 180,E1 -23559.414,E2 -23559.414} C_VEL
LIN {X 0,Y 157.752,Z 541.211,A -85,B 0,C 180,E1 -23564.497,E2 -23564.497} C_VEL
LIN {X 0,Y 157.518,Z 539.849,A -85,B 0,C 180,E1 -23566.454,E2 -23566.454} C_VEL
LIN {X 0,Y 157.722,Z 539.806,A -85,B 0,C 180,E1 -23569.733,E2 -23569.733} C_VEL
LIN {X 0,Y 157.781,Z 539.789,A -85,B 0,C 180,E1 -23572.321,E2 -23572.321} C_VEL
LIN {X 0,Y 158.254,Z 539.728,A -85,B 0,C 180,E1 -23580.001,E2 -23580.001} C_VEL
LIN {X 0,Y 157.765,Z 539.793,A -85,B 0,C 180,E1 -23587.681,E2 -23587.681} C_VEL
LIN {X 0,Y 157.641,Z 539.939,A -85,B 0,C 180,E1 -23591.442,E2 -23591.442} C_VEL
LIN {X 0,Y 158.438,Z 542.692,A -85,B 0,C 180,E1 -23595.436,E2 -23595.436} C_VEL
LIN {X 0,Y 159.597,Z 544.078,A -85,B 0,C 180,E1 -23597.955,E2 -23597.955} C_VEL
LIN {X 0,Y 161.721,Z 548.406,A -85,B 0,C 180,E1 -23603.025,E2 -23603.025} C_VEL
LIN {X 0,Y 164.036,Z 553.685,A -85,B 0,C 180,E1 -23607.945,E2 -23607.945} C_VEL
LIN {X 0,Y 169.338,Z 560.789,A -85,B 0,C 180,E1 -23611.6,E2 -23611.6} C_VEL
LIN {X 0,Y 173.678,Z 567.003,A -85,B 0,C 180,E1 -23614.22,E2 -23614.22} C_VEL
LIN {X 0,Y 176.611,Z 571.582,A -85,B 0,C 180,E1 -23615.854,E2 -23615.854} C_VEL
LIN {X 0,Y 181.396,Z 579.365,A -85,B 0,C 180,E1 -23618.31,E2 -23618.31} C_VEL
LIN {X 0,Y 187.004,Z 589.694,A -85,B 0,C 180,E1 -23620.954,E2 -23620.954} C_VEL
LIN {X 0,Y 192.529,Z 601.726,A -85,B 0,C 180,E1 -23623.388,E2 -23623.388} C_VEL
LIN {X 0,Y 194.748,Z 607.47,A -85,B 0,C 180,E1 -23624.346,E2 -23624.346} C_VEL
LIN {X 0,Y 190.988,Z 665.312,A -85,B 0,C 180,E1 -23626.283,E2 -23626.283} C_VEL
LIN {X 0,Y 189.397,Z 677.797,A -85,B 0,C 180,E1 -23627.013,E2 -23627.013} C_VEL
LIN {X 0,Y 187,Z 690.51,A -85,B 0,C 180,E1 -23628.158,E2 -23628.158} C_VEL
LIN {X 0,Y 184.245,Z 701.862,A -85,B 0,C 180,E1 -23629.575,E2 -23629.575} C_VEL
LIN {X 0,Y 181.297,Z 712.084,A -85,B 0,C 180,E1 -23631.265,E2 -23631.265} C_VEL
LIN {X 0,Y 177.325,Z 722.92,A -85,B 0,C 180,E1 -23633.524,E2 -23633.524} C_VEL
LIN {X 0,Y 173.328,Z 732.479,A -85,B 0,C 180,E1 -23636.116,E2 -23636.116} C_VEL
LIN {X 0,Y 169.689,Z 740.305,A -85,B 0,C 180,E1 -23638.822,E2 -23638.822} C_VEL
LIN {X 0,Y 165.779,Z 747.956,A -85,B 0,C 180,E1 -23642.204,E2 -23642.204} C_VEL
LIN {X 0,Y 162.616,Z 754.053,A -85,B 0,C 180,E1 -23645.76,E2 -23645.76} C_VEL
LIN {X 0,Y 159.966,Z 758.877,A -85,B 0,C 180,E1 -23649.423,E2 -23649.423} C_VEL
LIN {X 0,Y 157.752,Z 762.573,A -85,B 0,C 180,E1 -23653.168,E2 -23653.168} C_VEL
LIN {X 0,Y 156.296,Z 765.244,A -85,B 0,C 180,E1 -23657.007,E2 -23657.007} C_VEL
LIN {X 0,Y 155.115,Z 767.358,A -85,B 0,C 180,E1 -23662.188,E2 -23662.188} C_VEL
LIN {X 0,Y 154.855,Z 767.787,A -85,B 0,C 180,E1 -23664.792,E2 -23664.792} C_VEL
LIN {X 0,Y 154.747,Z 767.805,A -85,B 0,C 180,E1 -23667.669,E2 -23667.669} C_VEL
LIN {X 0,Y 154.984,Z 766.752,A -85,B 0,C 180,E1 -23672.599,E2 -23672.599} C_VEL
LIN {X 0,Y 155.613,Z 764.873,A -85,B 0,C 180,E1 -23676.482,E2 -23676.482} C_VEL
LIN {X 0,Y 157.097,Z 760.86,A -85,B 0,C 180,E1 -23681.614,E2 -23681.614} C_VEL
LIN {X 0,Y 158.892,Z 756.64,A -85,B 0,C 180,E1 -23685.39,E2 -23685.39} C_VEL
LIN {X 0,Y 161.311,Z 751.238,A -85,B 0,C 180,E1 -23689.072,E2 -23689.072} C_VEL
LIN {X 0,Y 164.256,Z 744.481,A -85,B 0,C 180,E1 -23692.648,E2 -23692.648} C_VEL
LIN {X 0,Y 167.768,Z 735.985,A -85,B 0,C 180,E1 -23696.094,E2 -23696.094} C_VEL
LIN {X 0,Y 171.059,Z 727.282,A -85,B 0,C 180,E1 -23698.864,E2 -23698.864} C_VEL
LIN {X 0,Y 174.802,Z 716.543,A -85,B 0,C 180,E1 -23701.511,E2 -23701.511} C_VEL
LIN {X 0,Y 178.003,Z 705.704,A -85,B 0,C 180,E1 -23703.555,E2 -23703.555} C_VEL
LIN {X 0,Y 180.743,Z 694.225,A -85,B 0,C 180,E1 -23705.229,E2 -23705.229} C_VEL
LIN {X 0,Y 182.938,Z 682.155,A -85,B 0,C 180,E1 -23706.545,E2 -23706.545} C_VEL
LIN {X 0,Y 184.679,Z 668.923,A -85,B 0,C 180,E1 -23707.508,E2 -23707.508} C_VEL
LIN {X 0,Y 185.774,Z 654.704,A -85,B 0,C 180,E1 -23708.114,E2 -23708.114} C_VEL
LIN {X 0,Y 188.83,Z 601.163,A -85,B 0,C 180,E1 -23709.96,E2 -23709.96} C_VEL
LIN {X 0,Y 185.377,Z 592.551,A -85,B 0,C 180,E1 -23711.339,E2 -23711.339} C_VEL
LIN {X 0,Y 182.49,Z 598.291,A -85,B 0,C 180,E1 -23711.869,E2 -23711.869} C_VEL
LIN {X 0,Y 179.856,Z 601.583,A -85,B 0,C 180,E1 -23712.477,E2 -23712.477} C_VEL
LIN {X 0,Y 177.836,Z 602.896,A -85,B 0,C 180,E1 -23713.027,E2 -23713.027} C_VEL
LIN {X 0,Y 177.057,Z 603.207,A -85,B 0,C 180,E1 -23713.255,E2 -23713.255} C_VEL
LIN {X 0,Y 173.295,Z 615.409,A -85,B 0,C 180,E1 -23713.779,E2 -23713.779} C_VEL
LIN {X 0,Y 170.488,Z 622.016,A -85,B 0,C 180,E1 -23714.336,E2 -23714.336} C_VEL
LIN {X 0,Y 168.729,Z 624.388,A -85,B 0,C 180,E1 -23714.803,E2 -23714.803} C_VEL
LIN {X 0,Y 167.462,Z 624.81,A -85,B 0,C 180,E1 -23715.226,E2 -23715.226} C_VEL
LIN {X 0,Y 166.603,Z 623.449,A -85,B 0,C 180,E1 -23715.62,E2 -23715.62} C_VEL
LIN {X 0,Y 166.152,Z 620.173,A -85,B 0,C 180,E1 -23716.021,E2 -23716.021} C_VEL
LIN {X 0,Y 165.096,Z 637.718,A -85,B 0,C 180,E1 -23717.328,E2 -23717.328} C_VEL
LIN {X 0,Y 163.776,Z 651.799,A -85,B 0,C 180,E1 -23718.92,E2 -23718.92} C_VEL
LIN {X 0,Y 162.321,Z 664.925,A -85,B 0,C 180,E1 -23720.933,E2 -23720.933} C_VEL
LIN {X 0,Y 160.641,Z 677.342,A -85,B 0,C 180,E1 -23723.409,E2 -23723.409} C_VEL
LIN {X 0,Y 159.115,Z 688.278,A -85,B 0,C 180,E1 -23726.145,E2 -23726.145} C_VEL
LIN {X 0,Y 157.665,Z 699.09,A -85,B 0,C 180,E1 -23729.532,E2 -23729.532} C_VEL
LIN {X 0,Y 156.478,Z 708.794,A -85,B 0,C 180,E1 -23733.311,E2 -23733.311} C_VEL
LIN {X 0,Y 155.699,Z 715.91,A -85,B 0,C 180,E1 -23736.736,E2 -23736.736} C_VEL
LIN {X 0,Y 155.214,Z 722.784,A -85,B 0,C 180,E1 -23740.835,E2 -23740.835} C_VEL
LIN {X 0,Y 155.268,Z 729.062,A -85,B 0,C 180,E1 -23745.584,E2 -23745.584} C_VEL
LIN {X 0,Y 156.008,Z 733.143,A -85,B 0,C 180,E1 -23749.618,E2 -23749.618} C_VEL
LIN {X 0,Y 156.815,Z 735.235,A -85,B 0,C 180,E1 -23752.272,E2 -23752.272} C_VEL
LIN {X 0,Y 159.337,Z 738.173,A -85,B 0,C 180,E1 -23757.471,E2 -23757.471} C_VEL
LIN {X 0,Y 161.655,Z 739.203,A -85,B 0,C 180,E1 -23760.773,E2 -23760.773} C_VEL
LIN {X 0,Y 165.376,Z 739.527,A -85,B 0,C 180,E1 -23764.875,E2 -23764.875} C_VEL
LIN {X 0,Y 170.87,Z 738.476,A -85,B 0,C 180,E1 -23769.469,E2 -23769.469} C_VEL
LIN {X 0,Y 173.983,Z 737.324,A -85,B 0,C 180,E1 -23771.652,E2 -23771.652} C_VEL
LIN {X 0,Y 181.082,Z 733.803,A -85,B 0,C 180,E1 -23775.764,E2 -23775.764} C_VEL
LIN {X 0,Y 187.071,Z 729.951,A -85,B 0,C 180,E1 -23778.622,E2 -23778.622} C_VEL
LIN {X 0,Y 193.61,Z 724.995,A -85,B 0,C 180,E1 -23781.284,E2 -23781.284} C_VEL
LIN {X 0,Y 200.552,Z 718.788,A -85,B 0,C 180,E1 -23783.797,E2 -23783.797} C_VEL
LIN {X 0,Y 207.866,Z 711.126,A -85,B 0,C 180,E1 -23786.074,E2 -23786.074} C_VEL
LIN {X 0,Y 215.007,Z 702.461,A -85,B 0,C 180,E1 -23788.05,E2 -23788.05} C_VEL
LIN {X 0,Y 221.715,Z 692.866,A -85,B 0,C 180,E1 -23789.725,E2 -23789.725} C_VEL
LIN {X 0,Y 228.475,Z 681.411,A -85,B 0,C 180,E1 -23791.271,E2 -23791.271} C_VEL
LIN {X 0,Y 234.197,Z 669.584,A -85,B 0,C 180,E1 -23792.488,E2 -23792.488} C_VEL
LIN {X 0,Y 238.803,Z 657.478,A -85,B 0,C 180,E1 -23793.445,E2 -23793.445} C_VEL
LIN {X 0,Y 242.607,Z 644.817,A -85,B 0,C 180,E1 -23794.192,E2 -23794.192} C_VEL
LIN {X 0,Y 243.58,Z 640.68,A -85,B 0,C 180,E1 -23794.397,E2 -23794.397} C_VEL
LIN {X 0,Y 243.199,Z 641.283,A -85,B 0,C 180,E1 -23796.461,E2 -23796.461} C_VEL
LIN {X 0,Y 242.968,Z 644.001,A -85,B 0,C 180,E1 -23798.57,E2 -23798.57} C_VEL
LIN {X 0,Y 239.627,Z 656.341,A -85,B 0,C 180,E1 -23799.09,E2 -23799.09} C_VEL
LIN {X 0,Y 237.736,Z 661.926,A -85,B 0,C 180,E1 -23799.194,E2 -23799.194} C_VEL
LIN {X 0,Y 233.857,Z 671.02,A -85,B 0,C 180,E1 -23798.981,E2 -23798.981} C_VEL
LIN {X 0,Y 229.434,Z 679.876,A -85,B 0,C 180,E1 -23798.828,E2 -23798.828} C_VEL
LIN {X 0,Y 226.681,Z 684.947,A -85,B 0,C 180,E1 -23799.039,E2 -23799.039} C_VEL
LIN {X 0,Y 220.306,Z 695.84,A -85,B 0,C 180,E1 -23800.039,E2 -23800.039} C_VEL
LIN {X 0,Y 212.804,Z 706.723,A -85,B 0,C 180,E1 -23801.366,E2 -23801.366} C_VEL
LIN {X 0,Y 204.484,Z 717.008,A -85,B 0,C 180,E1 -23803.086,E2 -23803.086} C_VEL
LIN {X 0,Y 196.45,Z 725.744,A -85,B 0,C 180,E1 -23805.046,E2 -23805.046} C_VEL
LIN {X 0,Y 188.898,Z 732.947,A -85,B 0,C 180,E1 -23807.236,E2 -23807.236} C_VEL
LIN {X 0,Y 180.665,Z 739.947,A -85,B 0,C 180,E1 -23810.07,E2 -23810.07} C_VEL
LIN {X 0,Y 172.183,Z 746.132,A -85,B 0,C 180,E1 -23813.713,E2 -23813.713} C_VEL
LIN {X 0,Y 166.541,Z 749.777,A -85,B 0,C 180,E1 -23816.73,E2 -23816.73} C_VEL
LIN {X 0,Y 160.137,Z 753.299,A -85,B 0,C 180,E1 -23821.135,E2 -23821.135} C_VEL
LIN {X 0,Y 155.067,Z 755.666,A -85,B 0,C 180,E1 -23825.928,E2 -23825.928} C_VEL
LIN {X 0,Y 152.253,Z 761.862,A -85,B 0,C 180,E1 -23829.745,E2 -23829.745} C_VEL
LIN {X 0,Y 150.038,Z 766.772,A -85,B 0,C 180,E1 -23833.678,E2 -23833.678} C_VEL
LIN {X 0,Y 148.687,Z 770.55,A -85,B 0,C 180,E1 -23837.72,E2 -23837.72} C_VEL
LIN {X 0,Y 147.911,Z 773.292,A -85,B 0,C 180,E1 -23841.805,E2 -23841.805} C_VEL
LIN {X 0,Y 147.689,Z 774.58,A -85,B 0,C 180,E1 -23844.539,E2 -23844.539} C_VEL
LIN {X 0,Y 147.638,Z 775.704,A -85,B 0,C 180,E1 -23848.5,E2 -23848.5} C_VEL
LIN {X 0,Y 147.65,Z 776.007,A -85,B 0,C 180,E1 -23851.671,E2 -23851.671} C_VEL
LIN {X 0,Y 147.69,Z 775.596,A -85,B 0,C 180,E1 -23855.461,E2 -23855.461} C_VEL
LIN {X 0,Y 147.918,Z 774.848,A -85,B 0,C 180,E1 -23858.195,E2 -23858.195} C_VEL
LIN {X 0,Y 148.417,Z 773.653,A -85,B 0,C 180,E1 -23860.918,E2 -23860.918} C_VEL
LIN {X 0,Y 149.638,Z 771.099,A -85,B 0,C 180,E1 -23864.97,E2 -23864.97} C_VEL
LIN {X 0,Y 151.554,Z 767.534,A -85,B 0,C 180,E1 -23868.941,E2 -23868.941} C_VEL
LIN {X 0,Y 154.229,Z 762.855,A -85,B 0,C 180,E1 -23872.788,E2 -23872.788} C_VEL
LIN {X 0,Y 157.545,Z 756.918,A -85,B 0,C 180,E1 -23876.493,E2 -23876.493} C_VEL
LIN {X 0,Y 161.313,Z 749.524,A -85,B 0,C 180,E1 -23880.067,E2 -23880.067} C_VEL
LIN {X 0,Y 165.04,Z 741.983,A -85,B 0,C 180,E1 -23882.883,E2 -23882.883} C_VEL
LIN {X 0,Y 169.23,Z 732.812,A -85,B 0,C 180,E1 -23885.549,E2 -23885.549} C_VEL
LIN {X 0,Y 173.298,Z 722.602,A -85,B 0,C 180,E1 -23887.834,E2 -23887.834} C_VEL
LIN {X 0,Y 177.131,Z 711.289,A -85,B 0,C 180,E1 -23889.775,E2 -23889.775} C_VEL
LIN {X 0,Y 180.441,Z 699.421,A -85,B 0,C 180,E1 -23891.276,E2 -23891.276} C_VEL
LIN {X 0,Y 183.185,Z 686.326,A -85,B 0,C 180,E1 -23892.453,E2 -23892.453} C_VEL
LIN {X 0,Y 185.086,Z 672.992,A -85,B 0,C 180,E1 -23893.227,E2 -23893.227} C_VEL
LIN {X 0,Y 188.343,Z 623.234,A -85,B 0,C 180,E1 -23894.952,E2 -23894.952} C_VEL
LIN {X 0,Y 187.04,Z 603.225,A -85,B 0,C 180,E1 -23896.462,E2 -23896.462} C_VEL
LIN {X 0,Y 186.354,Z 600.586,A -85,B 0,C 180,E1 -23896.839,E2 -23896.839} C_VEL
LIN {X 0,Y 183.92,Z 593.447,A -85,B 0,C 180,E1 -23898.092,E2 -23898.092} C_VEL
LIN {X 0,Y 178.582,Z 584.091,A -85,B 0,C 180,E1 -23900.689,E2 -23900.689} C_VEL
LIN {X 0,Y 173.398,Z 575.924,A -85,B 0,C 180,E1 -23903.466,E2 -23903.466} C_VEL
LIN {X 0,Y 169.62,Z 570.41,A -85,B 0,C 180,E1 -23905.699,E2 -23905.699} C_VEL
LIN {X 0,Y 164.157,Z 562.716,A -85,B 0,C 180,E1 -23909.367,E2 -23909.367} C_VEL
LIN {X 0,Y 158.881,Z 555.976,A -85,B 0,C 180,E1 -23913.747,E2 -23913.747} C_VEL
LIN {X 0,Y 158.193,Z 554.488,A -85,B 0,C 180,E1 -23915.036,E2 -23915.036} C_VEL
LIN {X 0,Y 156.146,Z 550.895,A -85,B 0,C 180,E1 -23918.896,E2 -23918.896} C_VEL
LIN {X 0,Y 153.352,Z 545.581,A -85,B 0,C 180,E1 -23926.754,E2 -23926.754} C_VEL
LIN {X 0,Y 152.063,Z 544.032,A -85,B 0,C 180,E1 -23932.031,E2 -23932.031} C_VEL
LIN {X 0,Y 151.862,Z 542.799,A -85,B 0,C 180,E1 -23940.001,E2 -23940.001} C_VEL
LIN {X 0,Y 153.147,Z 545.29,A -85,B 0,C 180,E1 -23950.578,E2 -23950.578} C_VEL
LIN {X 0,Y 155.317,Z 550.149,A -85,B 0,C 180,E1 -23958.467,E2 -23958.467} C_VEL
LIN {X 0,Y 157.299,Z 554.282,A -85,B 0,C 180,E1 -23963.188,E2 -23963.188} C_VEL
LIN {X 0,Y 162.411,Z 560.867,A -85,B 0,C 180,E1 -23967.548,E2 -23967.548} C_VEL
LIN {X 0,Y 166.822,Z 566.946,A -85,B 0,C 180,E1 -23970.719,E2 -23970.719} C_VEL
LIN {X 0,Y 170.813,Z 572.871,A -85,B 0,C 180,E1 -23973.264,E2 -23973.264} C_VEL
LIN {X 0,Y 175.475,Z 580.336,A -85,B 0,C 180,E1 -23975.945,E2 -23975.945} C_VEL
LIN {X 0,Y 181.281,Z 590.777,A -85,B 0,C 180,E1 -23978.962,E2 -23978.962} C_VEL
LIN {X 0,Y 186.869,Z 602.726,A -85,B 0,C 180,E1 -23981.639,E2 -23981.639} C_VEL
LIN {X 0,Y 189.635,Z 609.596,A -85,B 0,C 180,E1 -23982.91,E2 -23982.91} C_VEL
LIN {X 0,Y 185.79,Z 665.99,A -85,B 0,C 180,E1 -23984.826,E2 -23984.826} C_VEL
LIN {X 0,Y 183.988,Z 678.973,A -85,B 0,C 180,E1 -23985.614,E2 -23985.614} C_VEL
LIN {X 0,Y 181.515,Z 691.447,A -85,B 0,C 180,E1 -23986.779,E2 -23986.779} C_VEL
LIN {X 0,Y 178.571,Z 702.913,A -85,B 0,C 180,E1 -23988.255,E2 -23988.255} C_VEL
LIN {X 0,Y 175.287,Z 713.557,A -85,B 0,C 180,E1 -23990.097,E2 -23990.097} C_VEL
LIN {X 0,Y 171.22,Z 723.997,A -85,B 0,C 180,E1 -23992.37,E2 -23992.37} C_VEL
LIN {X 0,Y 166.671,Z 734.259,A -85,B 0,C 180,E1 -23995.303,E2 -23995.303} C_VEL
LIN {X 0,Y 162.201,Z 743.123,A -85,B 0,C 180,E1 -23998.672,E2 -23998.672} C_VEL
LIN {X 0,Y 158.323,Z 750.26,A -85,B 0,C 180,E1 -24002.221,E2 -24002.221} C_VEL
LIN {X 0,Y 155.118,Z 755.949,A -85,B 0,C 180,E1 -24005.936,E2 -24005.936} C_VEL
LIN {X 0,Y 152.467,Z 760.396,A -85,B 0,C 180,E1 -24009.775,E2 -24009.775} C_VEL
LIN {X 0,Y 150.356,Z 763.752,A -85,B 0,C 180,E1 -24013.713,E2 -24013.713} C_VEL
LIN {X 0,Y 149.37,Z 765.409,A -85,B 0,C 180,E1 -24016.394,E2 -24016.394} C_VEL
LIN {X 0,Y 148.061,Z 767.536,A -85,B 0,C 180,E1 -24021.813,E2 -24021.813} C_VEL
LIN {X 0,Y 147.769,Z 767.976,A -85,B 0,C 180,E1 -24024.542,E2 -24024.542} C_VEL
LIN {X 0,Y 147.653,Z 767.953,A -85,B 0,C 180,E1 -24028.329,E2 -24028.329} C_VEL
LIN {X 0,Y 147.895,Z 766.959,A -85,B 0,C 180,E1 -24032.724,E2 -24032.724} C_VEL
LIN {X 0,Y 148.416,Z 765.481,A -85,B 0,C 180,E1 -24036.047,E2 -24036.047} C_VEL
LIN {X 0,Y 149.668,Z 762.272,A -85,B 0,C 180,E1 -24040.826,E2 -24040.826} C_VEL
LIN {X 0,Y 151.347,Z 758.433,A -85,B 0,C 180,E1 -24044.797,E2 -24044.797} C_VEL
LIN {X 0,Y 153.699,Z 753.46,A -85,B 0,C 180,E1 -24048.667,E2 -24048.667} C_VEL
LIN {X 0,Y 156.65,Z 747.167,A -85,B 0,C 180,E1 -24052.417,E2 -24052.417} C_VEL
LIN {X 0,Y 160.08,Z 739.314,A -85,B 0,C 180,E1 -24056.041,E2 -24056.041} C_VEL
LIN {X 0,Y 163.479,Z 731.287,A -85,B 0,C 180,E1 -24058.923,E2 -24058.923} C_VEL
LIN {X 0,Y 167.236,Z 721.493,A -85,B 0,C 180,E1 -24061.688,E2 -24061.688} C_VEL
LIN {X 0,Y 170.909,Z 710.426,A -85,B 0,C 180,E1 -24064.074,E2 -24064.074} C_VEL
LIN {X 0,Y 173.845,Z 699.47,A -85,B 0,C 180,E1 -24065.919,E2 -24065.919} C_VEL
LIN {X 0,Y 176.452,Z 687.662,A -85,B 0,C 180,E1 -24067.401,E2 -24067.401} C_VEL
LIN {X 0,Y 178.43,Z 675.202,A -85,B 0,C 180,E1 -24068.521,E2 -24068.521} C_VEL
LIN {X 0,Y 179.86,Z 661.863,A -85,B 0,C 180,E1 -24069.277,E2 -24069.277} C_VEL
LIN {X 0,Y 183.221,Z 606.542,A -85,B 0,C 180,E1 -24071.226,E2 -24071.226} C_VEL
LIN {X 0,Y 180.886,Z 608.548,A -85,B 0,C 180,E1 -24071.796,E2 -24071.796} C_VEL
LIN {X 0,Y 177.06,Z 619.972,A -85,B 0,C 180,E1 -24072.328,E2 -24072.328} C_VEL
LIN {X 0,Y 174.339,Z 625.945,A -85,B 0,C 180,E1 -24072.844,E2 -24072.844} C_VEL
LIN {X 0,Y 171.669,Z 629.682,A -85,B 0,C 180,E1 -24073.494,E2 -24073.494} C_VEL
LIN {X 0,Y 169.309,Z 631.385,A -85,B 0,C 180,E1 -24074.185,E2 -24074.185} C_VEL
LIN {X 0,Y 168.331,Z 631.725,A -85,B 0,C 180,E1 -24074.502,E2 -24074.502} C_VEL
LIN {X 0,Y 165.107,Z 640.933,A -85,B 0,C 180,E1 -24075.086,E2 -24075.086} C_VEL
LIN {X 0,Y 162.201,Z 646.621,A -85,B 0,C 180,E1 -24075.804,E2 -24075.804} C_VEL
LIN {X 0,Y 160.045,Z 649.342,A -85,B 0,C 180,E1 -24076.457,E2 -24076.457} C_VEL
LIN {X 0,Y 158.515,Z 649.953,A -85,B 0,C 180,E1 -24077.024,E2 -24077.024} C_VEL
LIN {X 0,Y 157.858,Z 649.138,A -85,B 0,C 180,E1 -24077.346,E2 -24077.346} C_VEL
LIN {X 0,Y 157.434,Z 646.607,A -85,B 0,C 180,E1 -24077.692,E2 -24077.692} C_VEL
LIN {X 0,Y 157.41,Z 645.379,A -85,B 0,C 180,E1 -24077.792,E2 -24077.792} C_VEL
LIN {X 0,Y 155.961,Z 658.664,A -85,B 0,C 180,E1 -24079.618,E2 -24079.618} C_VEL
LIN {X 0,Y 154.506,Z 670.249,A -85,B 0,C 180,E1 -24081.7,E2 -24081.7} C_VEL
LIN {X 0,Y 152.883,Z 682.567,A -85,B 0,C 180,E1 -24084.523,E2 -24084.523} C_VEL
LIN {X 0,Y 151.257,Z 693.61,A -85,B 0,C 180,E1 -24087.7,E2 -24087.7} C_VEL
LIN {X 0,Y 149.942,Z 703.525,A -85,B 0,C 180,E1 -24091.285,E2 -24091.285} C_VEL
LIN {X 0,Y 149.046,Z 711.666,A -85,B 0,C 180,E1 -24094.888,E2 -24094.888} C_VEL
LIN {X 0,Y 148.3,Z 719.525,A -85,B 0,C 180,E1 -24099.18,E2 -24099.18} C_VEL
LIN {X 0,Y 148.084,Z 725.781,A -85,B 0,C 180,E1 -24103.455,E2 -24103.455} C_VEL
LIN {X 0,Y 148.488,Z 730.719,A -85,B 0,C 180,E1 -24107.702,E2 -24107.702} C_VEL
LIN {X 0,Y 149.534,Z 734.514,A -85,B 0,C 180,E1 -24111.894,E2 -24111.894} C_VEL
LIN {X 0,Y 152.004,Z 738.063,A -85,B 0,C 180,E1 -24117.349,E2 -24117.349} C_VEL
LIN {X 0,Y 154.647,Z 739.58,A -85,B 0,C 180,E1 -24121.224,E2 -24121.224} C_VEL
LIN {X 0,Y 158.097,Z 740.265,A -85,B 0,C 180,E1 -24125.1,E2 -24125.1} C_VEL
LIN {X 0,Y 163.728,Z 739.796,A -85,B 0,C 180,E1 -24129.886,E2 -24129.886} C_VEL
LIN {X 0,Y 166.92,Z 738.962,A -85,B 0,C 180,E1 -24132.152,E2 -24132.152} C_VEL
LIN {X 0,Y 174.23,Z 736.074,A -85,B 0,C 180,E1 -24136.401,E2 -24136.401} C_VEL
LIN {X 0,Y 180.398,Z 732.769,A -85,B 0,C 180,E1 -24139.338,E2 -24139.338} C_VEL
LIN {X 0,Y 187.066,Z 728.424,A -85,B 0,C 180,E1 -24142.067,E2 -24142.067} C_VEL
LIN {X 0,Y 195.244,Z 721.997,A -85,B 0,C 180,E1 -24144.964,E2 -24144.964} C_VEL
LIN {X 0,Y 203.046,Z 714.754,A -85,B 0,C 180,E1 -24147.298,E2 -24147.298} C_VEL
LIN {X 0,Y 210.651,Z 706.402,A -85,B 0,C 180,E1 -24149.327,E2 -24149.327} C_VEL
LIN {X 0,Y 217.975,Z 697.078,A -85,B 0,C 180,E1 -24151.056,E2 -24151.056} C_VEL
LIN {X 0,Y 224.503,Z 687.157,A -85,B 0,C 180,E1 -24152.469,E2 -24152.469} C_VEL
LIN {X 0,Y 231.147,Z 675.081,A -85,B 0,C 180,E1 -24153.799,E2 -24153.799} C_VEL
LIN {X 0,Y 236.732,Z 662.373,A -85,B 0,C 180,E1 -24154.861,E2 -24154.861} C_VEL
LIN {X 0,Y 241.042,Z 649.61,A -85,B 0,C 180,E1 -24155.671,E2 -24155.671} C_VEL
LIN {X 0,Y 241.529,Z 647.847,A -85,B 0,C 180,E1 -24155.788,E2 -24155.788} C_VEL
LIN {X 0,Y 241.306,Z 648.823,A -85,B 0,C 180,E1 -24156.829,E2 -24156.829} C_VEL
LIN {X 0,Y 241.171,Z 649.472,A -85,B 0,C 180,E1 -24157.094,E2 -24157.094} C_VEL
LIN {X 0,Y 236.772,Z 662.981,A -85,B 0,C 180,E1 -24157.674,E2 -24157.674} C_VEL
LIN {X 0,Y 231.008,Z 676.512,A -85,B 0,C 180,E1 -24158.429,E2 -24158.429} C_VEL
LIN {X 0,Y 226.681,Z 684.947,A -85,B 0,C 180,E1 -24159.039,E2 -24159.039} C_VEL
LIN {X 0,Y 223.734,Z 690.042,A -85,B 0,C 180,E1 -24159.298,E2 -24159.298} C_VEL
LIN {X 0,Y 218.13,Z 698.193,A -85,B 0,C 180,E1 -24159.367,E2 -24159.367} C_VEL
LIN {X 0,Y 212.081,Z 705.925,A -85,B 0,C 180,E1 -24159.523,E2 -24159.523} C_VEL
LIN {X 0,Y 208.45,Z 710.267,A -85,B 0,C 180,E1 -24159.934,E2 -24159.934} C_VEL
LIN {X 0,Y 199.833,Z 719.908,A -85,B 0,C 180,E1 -24161.64,E2 -24161.64} C_VEL
LIN {X 0,Y 190.288,Z 729.146,A -85,B 0,C 180,E1 -24163.93,E2 -24163.93} C_VEL
LIN {X 0,Y 182.612,Z 735.659,A -85,B 0,C 180,E1 -24166.153,E2 -24166.153} C_VEL
LIN {X 0,Y 175.352,Z 741.043,A -85,B 0,C 180,E1 -24168.601,E2 -24168.601} C_VEL
LIN {X 0,Y 168.651,Z 745.507,A -85,B 0,C 180,E1 -24171.313,E2 -24171.313} C_VEL
LIN {X 0,Y 160.663,Z 750.081,A -85,B 0,C 180,E1 -24175.344,E2 -24175.344} C_VEL
LIN {X 0,Y 153.95,Z 753.229,A -85,B 0,C 180,E1 -24179.858,E2 -24179.858} C_VEL
LIN {X 0,Y 148.732,Z 755.118,A -85,B 0,C 180,E1 -24184.646,E2 -24184.646} C_VEL
LIN {X 0,Y 145.584,Z 761.613,A -85,B 0,C 180,E1 -24188.774,E2 -24188.774} C_VEL
LIN {X 0,Y 143.201,Z 766.535,A -85,B 0,C 180,E1 -24192.875,E2 -24192.875} C_VEL
LIN {X 0,Y 141.722,Z 770.324,A -85,B 0,C 180,E1 -24197.106,E2 -24197.106} C_VEL
LIN {X 0,Y 140.858,Z 773.076,A -85,B 0,C 180,E1 -24201.392,E2 -24201.392} C_VEL
LIN {X 0,Y 140.618,Z 774.371,A -85,B 0,C 180,E1 -24204.263,E2 -24204.263} C_VEL
LIN {X 0,Y 140.578,Z 775.613,A -85,B 0,C 180,E1 -24209.065,E2 -24209.065} C_VEL
LIN {X 0,Y 140.547,Z 775.763,A -85,B 0,C 180,E1 -24212.866,E2 -24212.866} C_VEL
LIN {X 0,Y 140.619,Z 775.413,A -85,B 0,C 180,E1 -24215.737,E2 -24215.737} C_VEL
LIN {X 0,Y 140.866,Z 774.671,A -85,B 0,C 180,E1 -24218.608,E2 -24218.608} C_VEL
LIN {X 0,Y 141.424,Z 773.485,A -85,B 0,C 180,E1 -24221.465,E2 -24221.465} C_VEL
LIN {X 0,Y 142.737,Z 770.942,A -85,B 0,C 180,E1 -24225.712,E2 -24225.712} C_VEL
LIN {X 0,Y 144.847,Z 767.39,A -85,B 0,C 180,E1 -24229.854,E2 -24229.854} C_VEL
LIN {X 0,Y 147.669,Z 762.724,A -85,B 0,C 180,E1 -24233.862,E2 -24233.862} C_VEL
LIN {X 0,Y 151.179,Z 756.802,A -85,B 0,C 180,E1 -24237.702,E2 -24237.702} C_VEL
LIN {X 0,Y 155.183,Z 749.425,A -85,B 0,C 180,E1 -24241.386,E2 -24241.386} C_VEL
LIN {X 0,Y 159.122,Z 741.903,A -85,B 0,C 180,E1 -24244.272,E2 -24244.272} C_VEL
LIN {X 0,Y 163.509,Z 732.767,A -85,B 0,C 180,E1 -24246.994,E2 -24246.994} C_VEL
LIN {X 0,Y 167.746,Z 722.59,A -85,B 0,C 180,E1 -24249.322,E2 -24249.322} C_VEL
LIN {X 0,Y 171.747,Z 711.319,A -85,B 0,C 180,E1 -24251.287,E2 -24251.287} C_VEL
LIN {X 0,Y 175.179,Z 699.547,A -85,B 0,C 180,E1 -24252.804,E2 -24252.804} C_VEL
LIN {X 0,Y 178.019,Z 686.562,A -85,B 0,C 180,E1 -24253.993,E2 -24253.993} C_VEL
LIN {X 0,Y 180,Z 673.571,A -85,B 0,C 180,E1 -24254.767,E2 -24254.767} C_VEL
LIN {X 0,Y 183.394,Z 624.082,A -85,B 0,C 180,E1 -24256.518,E2 -24256.518} C_VEL
LIN {X 0,Y 182.334,Z 605.44,A -85,B 0,C 180,E1 -24257.961,E2 -24257.961} C_VEL
LIN {X 0,Y 179.926,Z 597.881,A -85,B 0,C 180,E1 -24259.305,E2 -24259.305} C_VEL
LIN {X 0,Y 174.528,Z 588.259,A -85,B 0,C 180,E1 -24262.119,E2 -24262.119} C_VEL
LIN {X 0,Y 168.416,Z 578.402,A -85,B 0,C 180,E1 -24265.714,E2 -24265.714} C_VEL
LIN {X 0,Y 161.628,Z 568.668,A -85,B 0,C 180,E1 -24270.431,E2 -24270.431} C_VEL
LIN {X 0,Y 155.606,Z 560.883,A -85,B 0,C 180,E1 -24275.661,E2 -24275.661} C_VEL
LIN {X 0,Y 151.476,Z 555.85,A -85,B 0,C 180,E1 -24280.344,E2 -24280.344} C_VEL
LIN {X 0,Y 149.502,Z 551.87,A -85,B 0,C 180,E1 -24286.406,E2 -24286.406} C_VEL
LIN {X 0,Y 148.143,Z 549.987,A -85,B 0,C 180,E1 -24291.818,E2 -24291.818} C_VEL
LIN {X 0,Y 147.832,Z 548.669,A -85,B 0,C 180,E1 -24300.001,E2 -24300.001} C_VEL
LIN {X 0,Y 148.393,Z 550.36,A -85,B 0,C 180,E1 -24308.169,E2 -24308.169} C_VEL
LIN {X 0,Y 148.975,Z 551.319,A -85,B 0,C 180,E1 -24310.878,E2 -24310.878} C_VEL
LIN {X 0,Y 150.483,Z 554.799,A -85,B 0,C 180,E1 -24316.587,E2 -24316.587} C_VEL
LIN {X 0,Y 152.219,Z 557.02,A -85,B 0,C 180,E1 -24318.857,E2 -24318.857} C_VEL
LIN {X 0,Y 155.564,Z 561.003,A -85,B 0,C 180,E1 -24322.495,E2 -24322.495} C_VEL
LIN {X 0,Y 160.091,Z 566.991,A -85,B 0,C 180,E1 -24326.567,E2 -24326.567} C_VEL
LIN {X 0,Y 164.475,Z 573.274,A -85,B 0,C 180,E1 -24329.899,E2 -24329.899} C_VEL
LIN {X 0,Y 169.224,Z 580.568,A -85,B 0,C 180,E1 -24333.042,E2 -24333.042} C_VEL
LIN {X 0,Y 174.751,Z 590.294,A -85,B 0,C 180,E1 -24336.296,E2 -24336.296} C_VEL
LIN {X 0,Y 179.567,Z 599.845,A -85,B 0,C 180,E1 -24338.862,E2 -24338.862} C_VEL
LIN {X 0,Y 184.347,Z 611.086,A -85,B 0,C 180,E1 -24341.257,E2 -24341.257} C_VEL
LIN {X 0,Y 184.617,Z 611.843,A -85,B 0,C 180,E1 -24341.392,E2 -24341.392} C_VEL
LIN {X 0,Y 180.762,Z 666.203,A -85,B 0,C 180,E1 -24343.265,E2 -24343.265} C_VEL
LIN {X 0,Y 178.953,Z 678.908,A -85,B 0,C 180,E1 -24344.042,E2 -24344.042} C_VEL
LIN {X 0,Y 176.151,Z 692.385,A -85,B 0,C 180,E1 -24345.317,E2 -24345.317} C_VEL
LIN {X 0,Y 172.862,Z 704.358,A -85,B 0,C 180,E1 -24346.922,E2 -24346.922} C_VEL
LIN {X 0,Y 168.943,Z 716.074,A -85,B 0,C 180,E1 -24349.066,E2 -24349.066} C_VEL
LIN {X 0,Y 164.719,Z 726.115,A -85,B 0,C 180,E1 -24351.392,E2 -24351.392} C_VEL
LIN {X 0,Y 160.03,Z 735.926,A -85,B 0,C 180,E1 -24354.417,E2 -24354.417} C_VEL
LIN {X 0,Y 155.406,Z 744.543,A -85,B 0,C 180,E1 -24357.902,E2 -24357.902} C_VEL
LIN {X 0,Y 151.426,Z 751.41,A -85,B 0,C 180,E1 -24361.594,E2 -24361.594} C_VEL
LIN {X 0,Y 147.671,Z 757.671,A -85,B 0,C 180,E1 -24366.139,E2 -24366.139} C_VEL
LIN {X 0,Y 144.927,Z 761.761,A -85,B 0,C 180,E1 -24370.157,E2 -24370.157} C_VEL
LIN {X 0,Y 143.508,Z 763.91,A -85,B 0,C 180,E1 -24372.913,E2 -24372.913} C_VEL
LIN {X 0,Y 142.45,Z 765.575,A -85,B 0,C 180,E1 -24375.719,E2 -24375.719} C_VEL
LIN {X 0,Y 141.029,Z 767.713,A -85,B 0,C 180,E1 -24381.402,E2 -24381.402} C_VEL
LIN {X 0,Y 140.704,Z 768.164,A -85,B 0,C 180,E1 -24384.267,E2 -24384.267} C_VEL
LIN {X 0,Y 140.581,Z 768.033,A -85,B 0,C 180,E1 -24389.065,E2 -24389.065} C_VEL
LIN {X 0,Y 140.826,Z 767.166,A -85,B 0,C 180,E1 -24392.86,E2 -24392.86} C_VEL
LIN {X 0,Y 141.263,Z 766.016,A -85,B 0,C 180,E1 -24395.71,E2 -24395.71} C_VEL
LIN {X 0,Y 141.888,Z 764.461,A -85,B 0,C 180,E1 -24398.545,E2 -24398.545} C_VEL
LIN {X 0,Y 143.232,Z 761.328,A -85,B 0,C 180,E1 -24402.756,E2 -24402.756} C_VEL
LIN {X 0,Y 145.275,Z 757.133,A -85,B 0,C 180,E1 -24406.873,E2 -24406.873} C_VEL
LIN {X 0,Y 148.455,Z 750.761,A -85,B 0,C 180,E1 -24411.524,E2 -24411.524} C_VEL
LIN {X 0,Y 151.892,Z 743.736,A -85,B 0,C 180,E1 -24415.34,E2 -24415.34} C_VEL
LIN {X 0,Y 155.825,Z 734.997,A -85,B 0,C 180,E1 -24419.002,E2 -24419.002} C_VEL
LIN {X 0,Y 159.604,Z 726.005,A -85,B 0,C 180,E1 -24421.897,E2 -24421.897} C_VEL
LIN {X 0,Y 163.334,Z 716.01,A -85,B 0,C 180,E1 -24424.384,E2 -24424.384} C_VEL
LIN {X 0,Y 166.666,Z 705.391,A -85,B 0,C 180,E1 -24426.453,E2 -24426.453} C_VEL
LIN {X 0,Y 169.73,Z 693.693,A -85,B 0,C 180,E1 -24428.178,E2 -24428.178} C_VEL
LIN {X 0,Y 172.107,Z 681.143,A -85,B 0,C 180,E1 -24429.55,E2 -24429.55} C_VEL
LIN {X 0,Y 173.932,Z 668.294,A -85,B 0,C 180,E1 -24430.468,E2 -24430.468} C_VEL
LIN {X 0,Y 175.322,Z 649.947,A -85,B 0,C 180,E1 -24431.218,E2 -24431.218} C_VEL
LIN {X 0,Y 176.406,Z 632.782,A -85,B 0,C 180,E1 -24431.827,E2 -24431.827} C_VEL
LIN {X 0,Y 173.331,Z 636.118,A -85,B 0,C 180,E1 -24432.592,E2 -24432.592} C_VEL
LIN {X 0,Y 171.795,Z 637.444,A -85,B 0,C 180,E1 -24433.007,E2 -24433.007} C_VEL
LIN {X 0,Y 168.715,Z 645.362,A -85,B 0,C 180,E1 -24433.563,E2 -24433.563} C_VEL
LIN {X 0,Y 165.471,Z 651.298,A -85,B 0,C 180,E1 -24434.323,E2 -24434.323} C_VEL
LIN {X 0,Y 162.471,Z 654.98,A -85,B 0,C 180,E1 -24435.175,E2 -24435.175} C_VEL
LIN {X 0,Y 159.879,Z 656.649,A -85,B 0,C 180,E1 -24436.047,E2 -24436.047} C_VEL
LIN {X 0,Y 158.281,Z 656.983,A -85,B 0,C 180,E1 -24436.652,E2 -24436.652} C_VEL
LIN {X 0,Y 154.906,Z 663.436,A -85,B 0,C 180,E1 -24437.555,E2 -24437.555} C_VEL
LIN {X 0,Y 151.812,Z 667.297,A -85,B 0,C 180,E1 -24438.534,E2 -24438.534} C_VEL
LIN {X 0,Y 150.304,Z 668.259,A -85,B 0,C 180,E1 -24439.108,E2 -24439.108} C_VEL
LIN {X 0,Y 148.91,Z 668.269,A -85,B 0,C 180,E1 -24439.758,E2 -24439.758} C_VEL
LIN {X 0,Y 148.327,Z 667.542,A -85,B 0,C 180,E1 -24440.122,E2 -24440.122} C_VEL
LIN {X 0,Y 148.108,Z 665.364,A -85,B 0,C 180,E1 -24440.494,E2 -24440.494} C_VEL
LIN {X 0,Y 146.226,Z 679.013,A -85,B 0,C 180,E1 -24443.502,E2 -24443.502} C_VEL
LIN {X 0,Y 144.622,Z 690.109,A -85,B 0,C 180,E1 -24446.625,E2 -24446.625} C_VEL
LIN {X 0,Y 143.1,Z 701.342,A -85,B 0,C 180,E1 -24450.585,E2 -24450.585} C_VEL
LIN {X 0,Y 142.105,Z 709.95,A -85,B 0,C 180,E1 -24454.357,E2 -24454.357} C_VEL
LIN {X 0,Y 141.302,Z 718.253,A -85,B 0,C 180,E1 -24458.862,E2 -24458.862} C_VEL
LIN {X 0,Y 141.022,Z 723.832,A -85,B 0,C 180,E1 -24462.601,E2 -24462.601} C_VEL
LIN {X 0,Y 141.305,Z 729.284,A -85,B 0,C 180,E1 -24467.066,E2 -24467.066} C_VEL
LIN {X 0,Y 142.257,Z 733.578,A -85,B 0,C 180,E1 -24471.476,E2 -24471.476} C_VEL
LIN {X 0,Y 143.308,Z 735.872,A -85,B 0,C 180,E1 -24474.371,E2 -24474.371} C_VEL
LIN {X 0,Y 144.675,Z 737.714,A -85,B 0,C 180,E1 -24477.215,E2 -24477.215} C_VEL
LIN {X 0,Y 148.45,Z 740.145,A -85,B 0,C 180,E1 -24482.713,E2 -24482.713} C_VEL
LIN {X 0,Y 153.554,Z 741.055,A -85,B 0,C 180,E1 -24487.891,E2 -24487.891} C_VEL
LIN {X 0,Y 159.841,Z 740.377,A -85,B 0,C 180,E1 -24492.699,E2 -24492.699} C_VEL
LIN {X 0,Y 167.36,Z 738.143,A -85,B 0,C 180,E1 -24497.094,E2 -24497.094} C_VEL
LIN {X 0,Y 173.682,Z 735.369,A -85,B 0,C 180,E1 -24500.117,E2 -24500.117} C_VEL
LIN {X 0,Y 180.492,Z 731.58,A -85,B 0,C 180,E1 -24502.916,E2 -24502.916} C_VEL
LIN {X 0,Y 188.864,Z 726.007,A -85,B 0,C 180,E1 -24505.818,E2 -24505.818} C_VEL
LIN {X 0,Y 196.914,Z 719.449,A -85,B 0,C 180,E1 -24508.223,E2 -24508.223} C_VEL
LIN {X 0,Y 205.354,Z 711.43,A -85,B 0,C 180,E1 -24510.386,E2 -24510.386} C_VEL
LIN {X 0,Y 212.272,Z 703.683,A -85,B 0,C 180,E1 -24511.987,E2 -24511.987} C_VEL
LIN {X 0,Y 220.736,Z 692.488,A -85,B 0,C 180,E1 -24513.741,E2 -24513.741} C_VEL
LIN {X 0,Y 227.826,Z 681.159,A -85,B 0,C 180,E1 -24515.068,E2 -24515.068} C_VEL
LIN {X 0,Y 232.899,Z 671.252,A -85,B 0,C 180,E1 -24515.978,E2 -24515.978} C_VEL
LIN {X 0,Y 232.43,Z 672.38,A -85,B 0,C 180,E1 -24516.417,E2 -24516.417} C_VEL
LIN {X 0,Y 226.076,Z 684.76,A -85,B 0,C 180,E1 -24517.195,E2 -24517.195} C_VEL
LIN {X 0,Y 219.047,Z 696.129,A -85,B 0,C 180,E1 -24518.182,E2 -24518.182} C_VEL
LIN {X 0,Y 209.97,Z 708.379,A -85,B 0,C 180,E1 -24519.662,E2 -24519.662} C_VEL
LIN {X 0,Y 208.45,Z 710.267,A -85,B 0,C 180,E1 -24519.934,E2 -24519.934} C_VEL
LIN {X 0,Y 204.617,Z 714.564,A -85,B 0,C 180,E1 -24520.41,E2 -24520.41} C_VEL
LIN {X 0,Y 197.49,Z 721.349,A -85,B 0,C 180,E1 -24520.873,E2 -24520.873} C_VEL
LIN {X 0,Y 190.152,Z 727.45,A -85,B 0,C 180,E1 -24521.505,E2 -24521.505} C_VEL
LIN {X 0,Y 186.045,Z 730.716,A -85,B 0,C 180,E1 -24522.258,E2 -24522.258} C_VEL
LIN {X 0,Y 177.648,Z 737.11,A -85,B 0,C 180,E1 -24524.595,E2 -24524.595} C_VEL
LIN {X 0,Y 170.159,Z 742.11,A -85,B 0,C 180,E1 -24527.041,E2 -24527.041} C_VEL
LIN {X 0,Y 161.027,Z 747.352,A -85,B 0,C 180,E1 -24530.74,E2 -24530.74} C_VEL
LIN {X 0,Y 154.894,Z 750.296,A -85,B 0,C 180,E1 -24533.855,E2 -24533.855} C_VEL
LIN {X 0,Y 147.837,Z 753.05,A -85,B 0,C 180,E1 -24538.472,E2 -24538.472} C_VEL
LIN {X 0,Y 142.481,Z 754.57,A -85,B 0,C 180,E1 -24543.264,E2 -24543.264} C_VEL
LIN {X 0,Y 139.87,Z 759.427,A -85,B 0,C 180,E1 -24546.299,E2 -24546.299} C_VEL
LIN {X 0,Y 137.179,Z 764.786,A -85,B 0,C 180,E1 -24550.549,E2 -24550.549} C_VEL
LIN {X 0,Y 135.238,Z 768.954,A -85,B 0,C 180,E1 -24554.94,E2 -24554.94} C_VEL
LIN {X 0,Y 134.418,Z 771.154,A -85,B 0,C 180,E1 -24557.928,E2 -24557.928} C_VEL
LIN {X 0,Y 133.828,Z 772.862,A -85,B 0,C 180,E1 -24560.936,E2 -24560.936} C_VEL
LIN {X 0,Y 133.543,Z 774.161,A -85,B 0,C 180,E1 -24563.958,E2 -24563.958} C_VEL
LIN {X 0,Y 133.466,Z 775.063,A -85,B 0,C 180,E1 -24566.982,E2 -24566.982} C_VEL
LIN {X 0,Y 133.531,Z 775.531,A -85,B 0,C 180,E1 -24570,E2 -24570} C_VEL
LIN {X 0,Y 133.466,Z 775.575,A -85,B 0,C 180,E1 -24573.018,E2 -24573.018} C_VEL
LIN {X 0,Y 133.544,Z 775.229,A -85,B 0,C 180,E1 -24576.042,E2 -24576.042} C_VEL
LIN {X 0,Y 133.838,Z 774.494,A -85,B 0,C 180,E1 -24579.064,E2 -24579.064} C_VEL
LIN {X 0,Y 134.456,Z 773.317,A -85,B 0,C 180,E1 -24582.068,E2 -24582.068} C_VEL
LIN {X 0,Y 135.876,Z 770.785,A -85,B 0,C 180,E1 -24586.527,E2 -24586.527} C_VEL
LIN {X 0,Y 138.155,Z 767.246,A -85,B 0,C 180,E1 -24590.86,E2 -24590.86} C_VEL
LIN {X 0,Y 141.178,Z 762.593,A -85,B 0,C 180,E1 -24595.032,E2 -24595.032} C_VEL
LIN {X 0,Y 144.871,Z 756.685,A -85,B 0,C 180,E1 -24599.02,E2 -24599.02} C_VEL
LIN {X 0,Y 149.161,Z 749.326,A -85,B 0,C 180,E1 -24602.808,E2 -24602.808} C_VEL
LIN {X 0,Y 153.314,Z 741.824,A -85,B 0,C 180,E1 -24605.764,E2 -24605.764} C_VEL
LIN {X 0,Y 157.893,Z 732.72,A -85,B 0,C 180,E1 -24608.546,E2 -24608.546} C_VEL
LIN {X 0,Y 162.308,Z 722.578,A -85,B 0,C 180,E1 -24610.912,E2 -24610.912} C_VEL
LIN {X 0,Y 166.47,Z 711.35,A -85,B 0,C 180,E1 -24612.902,E2 -24612.902} C_VEL
LIN {X 0,Y 170.053,Z 699.667,A -85,B 0,C 180,E1 -24614.425,E2 -24614.425} C_VEL
LIN {X 0,Y 173.004,Z 686.797,A -85,B 0,C 180,E1 -24615.619,E2 -24615.619} C_VEL
LIN {X 0,Y 175.123,Z 673.399,A -85,B 0,C 180,E1 -24616.433,E2 -24616.433} C_VEL
LIN {X 0,Y 178.601,Z 624.636,A -85,B 0,C 180,E1 -24618.184,E2 -24618.184} C_VEL
LIN {X 0,Y 177.775,Z 608.089,A -85,B 0,C 180,E1 -24619.506,E2 -24619.506} C_VEL
LIN {X 0,Y 175.98,Z 602.315,A -85,B 0,C 180,E1 -24620.586,E2 -24620.586} C_VEL
LIN {X 0,Y 170.747,Z 592.739,A -85,B 0,C 180,E1 -24623.519,E2 -24623.519} C_VEL
LIN {X 0,Y 164.894,Z 583.146,A -85,B 0,C 180,E1 -24627.233,E2 -24627.233} C_VEL
LIN {X 0,Y 159.114,Z 574.577,A -85,B 0,C 180,E1 -24631.563,E2 -24631.563} C_VEL
LIN {X 0,Y 153.815,Z 567.42,A -85,B 0,C 180,E1 -24636.462,E2 -24636.462} C_VEL
LIN {X 0,Y 149.835,Z 562.446,A -85,B 0,C 180,E1 -24641.188,E2 -24641.188} C_VEL
LIN {X 0,Y 146.12,Z 557.87,A -85,B 0,C 180,E1 -24647.501,E2 -24647.501} C_VEL
LIN {X 0,Y 144.383,Z 555.979,A -85,B 0,C 180,E1 -24652.308,E2 -24652.308} C_VEL
LIN {X 0,Y 143.833,Z 554.537,A -85,B 0,C 180,E1 -24660.001,E2 -24660.001} C_VEL
LIN {X 0,Y 144.067,Z 555.628,A -85,B 0,C 180,E1 -24664.547,E2 -24664.547} C_VEL
LIN {X 0,Y 145.559,Z 557.228,A -85,B 0,C 180,E1 -24669.379,E2 -24669.379} C_VEL
LIN {X 0,Y 147.037,Z 559.265,A -85,B 0,C 180,E1 -24672.597,E2 -24672.597} C_VEL
LIN {X 0,Y 150.07,Z 562.745,A -85,B 0,C 180,E1 -24677.311,E2 -24677.311} C_VEL
LIN {X 0,Y 153.714,Z 567.445,A -85,B 0,C 180,E1 -24681.632,E2 -24681.632} C_VEL
LIN {X 0,Y 157.994,Z 573.335,A -85,B 0,C 180,E1 -24685.706,E2 -24685.706} C_VEL
LIN {X 0,Y 162.378,Z 579.908,A -85,B 0,C 180,E1 -24689.214,E2 -24689.214} C_VEL
LIN {X 0,Y 166.616,Z 586.858,A -85,B 0,C 180,E1 -24692.178,E2 -24692.178} C_VEL
LIN {X 0,Y 171.565,Z 595.896,A -85,B 0,C 180,E1 -24695.264,E2 -24695.264} C_VEL
LIN {X 0,Y 175.666,Z 604.322,A -85,B 0,C 180,E1 -24697.599,E2 -24697.599} C_VEL
LIN {X 0,Y 179.794,Z 614.352,A -85,B 0,C 180,E1 -24699.827,E2 -24699.827} C_VEL
LIN {X 0,Y 175.89,Z 666.324,A -85,B 0,C 180,E1 -24701.614,E2 -24701.614} C_VEL
LIN {X 0,Y 174.006,Z 679.094,A -85,B 0,C 180,E1 -24702.397,E2 -24702.397} C_VEL
LIN {X 0,Y 171.177,Z 692.24,A -85,B 0,C 180,E1 -24703.647,E2 -24703.647} C_VEL
LIN {X 0,Y 167.798,Z 704.089,A -85,B 0,C 180,E1 -24705.221,E2 -24705.221} C_VEL
LIN {X 0,Y 164.118,Z 714.813,A -85,B 0,C 180,E1 -24707.172,E2 -24707.172} C_VEL
LIN {X 0,Y 159.713,Z 725.108,A -85,B 0,C 180,E1 -24709.531,E2 -24709.531} C_VEL
LIN {X 0,Y 155.177,Z 734.394,A -85,B 0,C 180,E1 -24712.309,E2 -24712.309} C_VEL
LIN {X 0,Y 150.21,Z 743.306,A -85,B 0,C 180,E1 -24715.845,E2 -24715.845} C_VEL
LIN {X 0,Y 145.824,Z 750.478,A -85,B 0,C 180,E1 -24719.6,E2 -24719.6} C_VEL
LIN {X 0,Y 142.21,Z 756.206,A -85,B 0,C 180,E1 -24723.592,E2 -24723.592} C_VEL
LIN {X 0,Y 139.206,Z 760.684,A -85,B 0,C 180,E1 -24727.751,E2 -24727.751} C_VEL
LIN {X 0,Y 136.697,Z 764.068,A -85,B 0,C 180,E1 -24732.033,E2 -24732.033} C_VEL
LIN {X 0,Y 135.538,Z 765.741,A -85,B 0,C 180,E1 -24734.974,E2 -24734.974} C_VEL
LIN {X 0,Y 133.996,Z 767.891,A -85,B 0,C 180,E1 -24740.947,E2 -24740.947} C_VEL
LIN {X 0,Y 133.638,Z 768.352,A -85,B 0,C 180,E1 -24743.963,E2 -24743.963} C_VEL
LIN {X 0,Y 133.491,Z 768.403,A -85,B 0,C 180,E1 -24746.982,E2 -24746.982} C_VEL
LIN {X 0,Y 133.534,Z 768.077,A -85,B 0,C 180,E1 -24750,E2 -24750} C_VEL
LIN {X 0,Y 133.95,Z 766.838,A -85,B 0,C 180,E1 -24754.512,E2 -24754.512} C_VEL
LIN {X 0,Y 134.875,Z 764.683,A -85,B 0,C 180,E1 -24758.993,E2 -24758.993} C_VEL
LIN {X 0,Y 136.328,Z 761.562,A -85,B 0,C 180,E1 -24763.414,E2 -24763.414} C_VEL
LIN {X 0,Y 138.508,Z 757.38,A -85,B 0,C 180,E1 -24767.724,E2 -24767.724} C_VEL
LIN {X 0,Y 141.878,Z 751.025,A -85,B 0,C 180,E1 -24772.575,E2 -24772.575} C_VEL
LIN {X 0,Y 145.532,Z 744.018,A -85,B 0,C 180,E1 -24776.531,E2 -24776.531} C_VEL
LIN {X 0,Y 148.958,Z 736.887,A -85,B 0,C 180,E1 -24779.695,E2 -24779.695} C_VEL
LIN {X 0,Y 152.829,Z 728.242,A -85,B 0,C 180,E1 -24782.706,E2 -24782.706} C_VEL
LIN {X 0,Y 157.116,Z 717.612,A -85,B 0,C 180,E1 -24785.556,E2 -24785.556} C_VEL
LIN {X 0,Y 160.742,Z 706.89,A -85,B 0,C 180,E1 -24787.741,E2 -24787.741} C_VEL
LIN {X 0,Y 163.895,Z 695.493,A -85,B 0,C 180,E1 -24789.518,E2 -24789.518} C_VEL
LIN {X 0,Y 166.54,Z 682.858,A -85,B 0,C 180,E1 -24790.989,E2 -24790.989} C_VEL
LIN {X 0,Y 168.471,Z 670.174,A -85,B 0,C 180,E1 -24791.96,E2 -24791.96} C_VEL
LIN {X 0,Y 169.739,Z 655.966,A -85,B 0,C 180,E1 -24792.611,E2 -24792.611} C_VEL
LIN {X 0,Y 169.757,Z 654.62,A -85,B 0,C 180,E1 -24792.682,E2 -24792.682} C_VEL
LIN {X 0,Y 166.056,Z 659.5,A -85,B 0,C 180,E1 -24793.625,E2 -24793.625} C_VEL
LIN {X 0,Y 162.804,Z 662.267,A -85,B 0,C 180,E1 -24794.578,E2 -24794.578} C_VEL
LIN {X 0,Y 160.654,Z 663.52,A -85,B 0,C 180,E1 -24795.265,E2 -24795.265} C_VEL
LIN {X 0,Y 156.886,Z 669.4,A -85,B 0,C 180,E1 -24796.162,E2 -24796.162} C_VEL
LIN {X 0,Y 153.301,Z 673.222,A -85,B 0,C 180,E1 -24797.18,E2 -24797.18} C_VEL
LIN {X 0,Y 150.444,Z 674.896,A -85,B 0,C 180,E1 -24798.174,E2 -24798.174} C_VEL
LIN {X 0,Y 147.435,Z 675.511,A -85,B 0,C 180,E1 -24799.465,E2 -24799.465} C_VEL
LIN {X 0,Y 144.197,Z 679.125,A -85,B 0,C 180,E1 -24800.456,E2 -24800.456} C_VEL
LIN {X 0,Y 141.371,Z 680.872,A -85,B 0,C 180,E1 -24801.579,E2 -24801.579} C_VEL
LIN {X 0,Y 139.836,Z 680.719,A -85,B 0,C 180,E1 -24802.454,E2 -24802.454} C_VEL
LIN {X 0,Y 139.246,Z 679.528,A -85,B 0,C 180,E1 -24803.042,E2 -24803.042} C_VEL
LIN {X 0,Y 139.156,Z 678.695,A -85,B 0,C 180,E1 -24803.333,E2 -24803.333} C_VEL
LIN {X 0,Y 137.477,Z 690.142,A -85,B 0,C 180,E1 -24806.663,E2 -24806.663} C_VEL
LIN {X 0,Y 136.025,Z 700.786,A -85,B 0,C 180,E1 -24810.554,E2 -24810.554} C_VEL
LIN {X 0,Y 135.014,Z 709.666,A -85,B 0,C 180,E1 -24814.567,E2 -24814.567} C_VEL
LIN {X 0,Y 134.23,Z 717.806,A -85,B 0,C 180,E1 -24819.153,E2 -24819.153} C_VEL
LIN {X 0,Y 133.998,Z 724.754,A -85,B 0,C 180,E1 -24824.016,E2 -24824.016} C_VEL
LIN {X 0,Y 134.644,Z 730.963,A -85,B 0,C 180,E1 -24829.473,E2 -24829.473} C_VEL
LIN {X 0,Y 135.991,Z 734.979,A -85,B 0,C 180,E1 -24834.067,E2 -24834.067} C_VEL
LIN {X 0,Y 137.334,Z 737.12,A -85,B 0,C 180,E1 -24837.066,E2 -24837.066} C_VEL
LIN {X 0,Y 141.126,Z 740.156,A -85,B 0,C 180,E1 -24842.854,E2 -24842.854} C_VEL
LIN {X 0,Y 146.304,Z 741.654,A -85,B 0,C 180,E1 -24848.285,E2 -24848.285} C_VEL
LIN {X 0,Y 152.745,Z 741.571,A -85,B 0,C 180,E1 -24853.3,E2 -24853.3} C_VEL
LIN {X 0,Y 160.481,Z 739.988,A -85,B 0,C 180,E1 -24857.851,E2 -24857.851} C_VEL
LIN {X 0,Y 164.714,Z 738.593,A -85,B 0,C 180,E1 -24859.958,E2 -24859.958} C_VEL
LIN {X 0,Y 173.973,Z 734.514,A -85,B 0,C 180,E1 -24863.826,E2 -24863.826} C_VEL
LIN {X 0,Y 182.497,Z 729.642,A -85,B 0,C 180,E1 -24866.751,E2 -24866.751} C_VEL
LIN {X 0,Y 190.844,Z 723.844,A -85,B 0,C 180,E1 -24869.205,E2 -24869.205} C_VEL
LIN {X 0,Y 199.205,Z 716.902,A -85,B 0,C 180,E1 -24871.318,E2 -24871.318} C_VEL
LIN {X 0,Y 208.071,Z 708.206,A -85,B 0,C 180,E1 -24873.29,E2 -24873.29} C_VEL
